PROGRAM C20_ProfinetDrivesCtrl
VAR

	(*G_xLabellerSemaLock	: BOOL;		(* This needs to be used to make sure only 1 client is using the FB instance *)

	fbParameterDisplay		: ARRAY[1..cMAX_PROFINET_DRIVES] OF FB_ParameterDisplayWrapper;
							aProfiNetDrives         : ARRAY[1..cMAX_PROFINET_DRIVES] OF ST_ParameterControl;____					
	xModuleIsActive			: ARRAY[1..cMAX_PROFINET_DRIVES] OF BOOL;*)

	fbProfinetCtrl			: ARRAY[1..cMAX_PROFINET_DRIVES] OF FB_G120Simple_V001;

(*dummy sturcture to be replaced by global PROFINET struct once implemnted*)
{library private}
	stEmptyDriveIn								: ST_DRIVE_INPUT;
	stEmptyDriveOut								: ST_DRIVE_OUTPUT;
	nNoCheckPNetIoError							: UINT;
END_VAR
VAR // added by the converter: edge detectors and wires of the graphical bodies
    _w1, _w2 : BOOL;
END_VAR

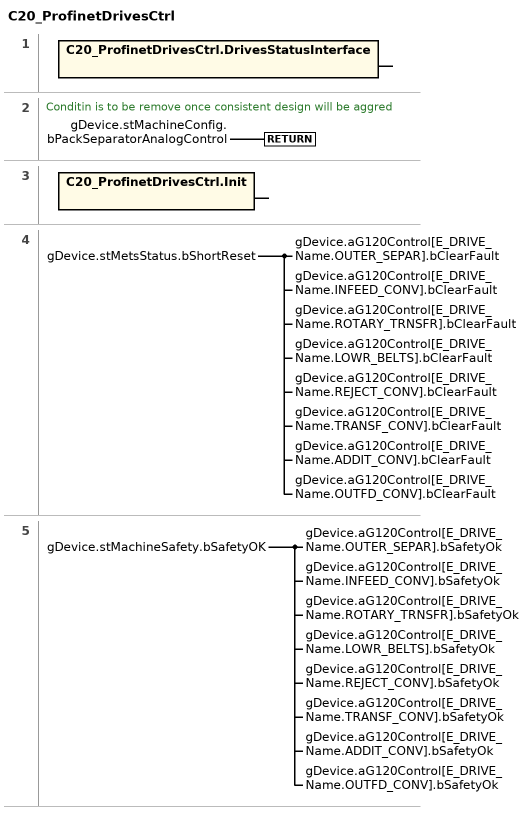
// NETWORK 1
C20_ProfinetDrivesCtrl.DrivesStatusInterface();

// NETWORK 2
// Conditin is to be remove once consistent design will be aggred
IF gDevice.stMachineConfig.bPackSeparatorAnalogControl THEN RETURN; END_IF

// NETWORK 3
C20_ProfinetDrivesCtrl.Init();

// NETWORK 4
_w1 := gDevice.stMetsStatus.bShortReset;
gDevice.aG120Control[E_DRIVE_Name.OUTER_SEPAR].bClearFault := _w1;
gDevice.aG120Control[E_DRIVE_Name.INFEED_CONV].bClearFault := _w1;
gDevice.aG120Control[E_DRIVE_Name.ROTARY_TRNSFR].bClearFault := _w1;
gDevice.aG120Control[E_DRIVE_Name.LOWR_BELTS].bClearFault := _w1;
gDevice.aG120Control[E_DRIVE_Name.REJECT_CONV].bClearFault := _w1;
gDevice.aG120Control[E_DRIVE_Name.TRANSF_CONV].bClearFault := _w1;
gDevice.aG120Control[E_DRIVE_Name.ADDIT_CONV].bClearFault := _w1;
gDevice.aG120Control[E_DRIVE_Name.OUTFD_CONV].bClearFault := _w1;

// NETWORK 5
_w2 := gDevice.stMachineSafety.bSafetyOK;
gDevice.aG120Control[E_DRIVE_Name.OUTER_SEPAR].bSafetyOk := _w2;
gDevice.aG120Control[E_DRIVE_Name.INFEED_CONV].bSafetyOk := _w2;
gDevice.aG120Control[E_DRIVE_Name.ROTARY_TRNSFR].bSafetyOk := _w2;
gDevice.aG120Control[E_DRIVE_Name.LOWR_BELTS].bSafetyOk := _w2;
gDevice.aG120Control[E_DRIVE_Name.REJECT_CONV].bSafetyOk := _w2;
gDevice.aG120Control[E_DRIVE_Name.TRANSF_CONV].bSafetyOk := _w2;
gDevice.aG120Control[E_DRIVE_Name.ADDIT_CONV].bSafetyOk := _w2;
gDevice.aG120Control[E_DRIVE_Name.OUTFD_CONV].bSafetyOk := _w2;

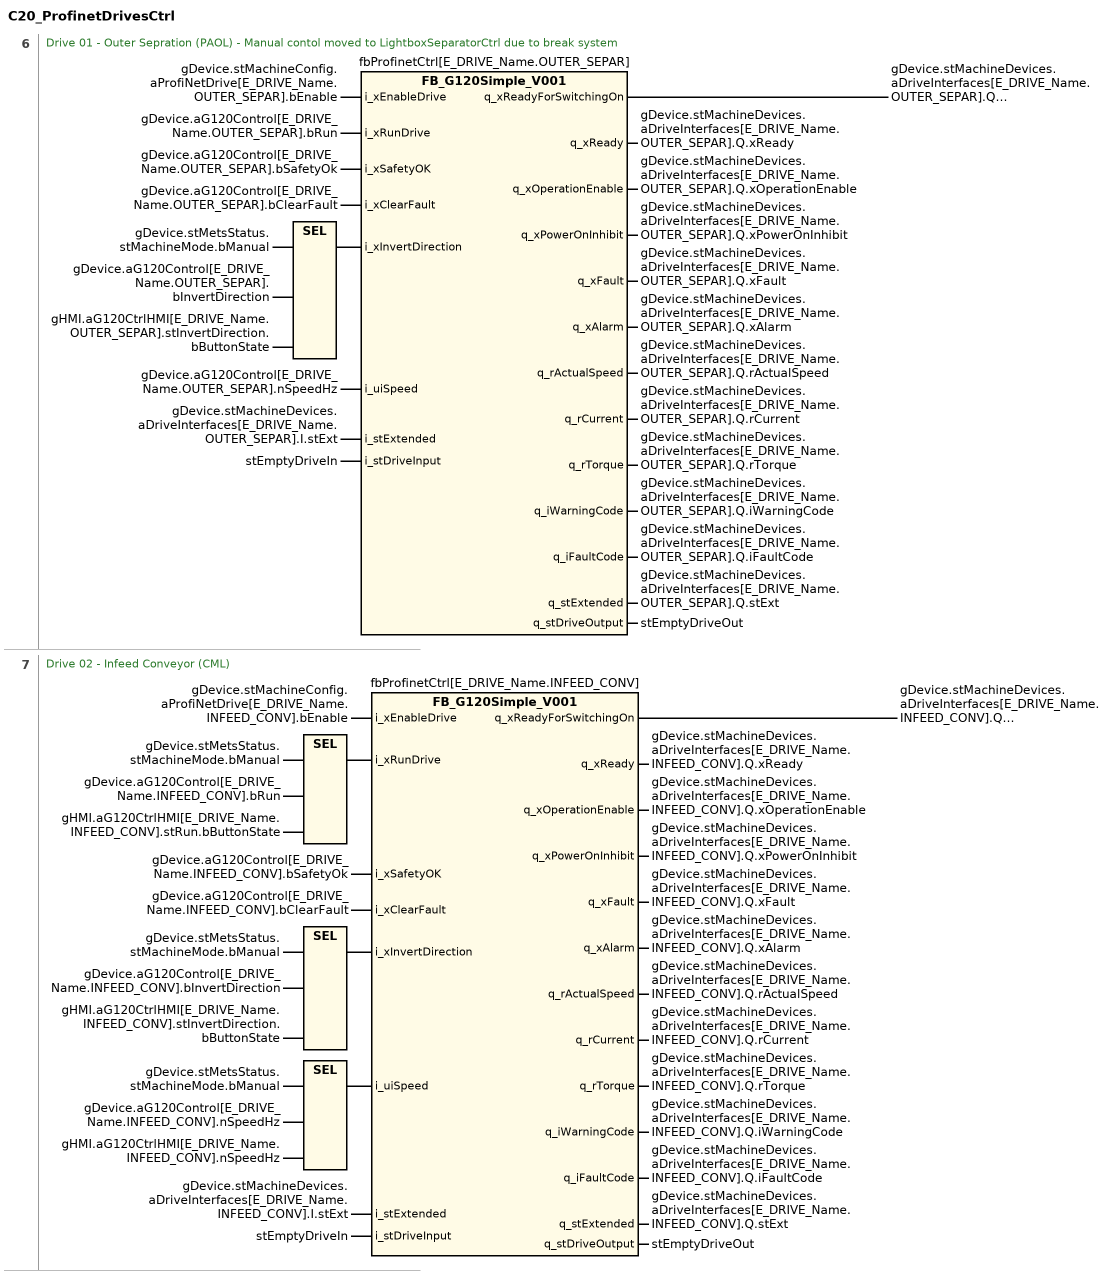
// NETWORK 6
// Drive 01 - Outer Sepration (PAOL) - Manual contol moved to LightboxSeparatorCtrl due to break system
fbProfinetCtrl[E_DRIVE_Name.OUTER_SEPAR](
    i_xEnableDrive := gDevice.stMachineConfig.aProfiNetDrive[E_DRIVE_Name.OUTER_SEPAR].bEnable,
    i_xRunDrive := gDevice.aG120Control[E_DRIVE_Name.OUTER_SEPAR].bRun,
    i_xSafetyOK := gDevice.aG120Control[E_DRIVE_Name.OUTER_SEPAR].bSafetyOk,
    i_xClearFault := gDevice.aG120Control[E_DRIVE_Name.OUTER_SEPAR].bClearFault,
    i_xInvertDirection := SEL(gDevice.stMetsStatus.stMachineMode.bManual, gDevice.aG120Control[E_DRIVE_Name.OUTER_SEPAR].bInvertDirection, gHMI.aG120CtrlHMI[E_DRIVE_Name.OUTER_SEPAR].stInvertDirection.bButtonState),
    i_uiSpeed := gDevice.aG120Control[E_DRIVE_Name.OUTER_SEPAR].nSpeedHz,
    i_stExtended := gDevice.stMachineDevices.aDriveInterfaces[E_DRIVE_Name.OUTER_SEPAR].I.stExt,
    i_stDriveInput := stEmptyDriveIn,
    q_xReady => gDevice.stMachineDevices.aDriveInterfaces[E_DRIVE_Name.OUTER_SEPAR].Q.xReady,
    q_xOperationEnable => gDevice.stMachineDevices.aDriveInterfaces[E_DRIVE_Name.OUTER_SEPAR].Q.xOperationEnable,
    q_xPowerOnInhibit => gDevice.stMachineDevices.aDriveInterfaces[E_DRIVE_Name.OUTER_SEPAR].Q.xPowerOnInhibit,
    q_xFault => gDevice.stMachineDevices.aDriveInterfaces[E_DRIVE_Name.OUTER_SEPAR].Q.xFault,
    q_xAlarm => gDevice.stMachineDevices.aDriveInterfaces[E_DRIVE_Name.OUTER_SEPAR].Q.xAlarm,
    q_rActualSpeed => gDevice.stMachineDevices.aDriveInterfaces[E_DRIVE_Name.OUTER_SEPAR].Q.rActualSpeed,
    q_rCurrent => gDevice.stMachineDevices.aDriveInterfaces[E_DRIVE_Name.OUTER_SEPAR].Q.rCurrent,
    q_rTorque => gDevice.stMachineDevices.aDriveInterfaces[E_DRIVE_Name.OUTER_SEPAR].Q.rTorque,
    q_iWarningCode => gDevice.stMachineDevices.aDriveInterfaces[E_DRIVE_Name.OUTER_SEPAR].Q.iWarningCode,
    q_iFaultCode => gDevice.stMachineDevices.aDriveInterfaces[E_DRIVE_Name.OUTER_SEPAR].Q.iFaultCode,
    q_stExtended => gDevice.stMachineDevices.aDriveInterfaces[E_DRIVE_Name.OUTER_SEPAR].Q.stExt,
    q_stDriveOutput => stEmptyDriveOut); // FB_G120Simple_V001
gDevice.stMachineDevices.aDriveInterfaces[E_DRIVE_Name.OUTER_SEPAR].Q.xReadyForSwitchingOn := fbProfinetCtrl[E_DRIVE_Name.OUTER_SEPAR].q_xReadyForSwitchingOn;

// NETWORK 7
// Drive 02 - Infeed Conveyor (CML)
fbProfinetCtrl[E_DRIVE_Name.INFEED_CONV](
    i_xEnableDrive := gDevice.stMachineConfig.aProfiNetDrive[E_DRIVE_Name.INFEED_CONV].bEnable,
    i_xRunDrive := SEL(gDevice.stMetsStatus.stMachineMode.bManual, gDevice.aG120Control[E_DRIVE_Name.INFEED_CONV].bRun, gHMI.aG120CtrlHMI[E_DRIVE_Name.INFEED_CONV].stRun.bButtonState),
    i_xSafetyOK := gDevice.aG120Control[E_DRIVE_Name.INFEED_CONV].bSafetyOk,
    i_xClearFault := gDevice.aG120Control[E_DRIVE_Name.INFEED_CONV].bClearFault,
    i_xInvertDirection := SEL(gDevice.stMetsStatus.stMachineMode.bManual, gDevice.aG120Control[E_DRIVE_Name.INFEED_CONV].bInvertDirection, gHMI.aG120CtrlHMI[E_DRIVE_Name.INFEED_CONV].stInvertDirection.bButtonState),
    i_uiSpeed := SEL(gDevice.stMetsStatus.stMachineMode.bManual, gDevice.aG120Control[E_DRIVE_Name.INFEED_CONV].nSpeedHz, gHMI.aG120CtrlHMI[E_DRIVE_Name.INFEED_CONV].nSpeedHz),
    i_stExtended := gDevice.stMachineDevices.aDriveInterfaces[E_DRIVE_Name.INFEED_CONV].I.stExt,
    i_stDriveInput := stEmptyDriveIn,
    q_xReady => gDevice.stMachineDevices.aDriveInterfaces[E_DRIVE_Name.INFEED_CONV].Q.xReady,
    q_xOperationEnable => gDevice.stMachineDevices.aDriveInterfaces[E_DRIVE_Name.INFEED_CONV].Q.xOperationEnable,
    q_xPowerOnInhibit => gDevice.stMachineDevices.aDriveInterfaces[E_DRIVE_Name.INFEED_CONV].Q.xPowerOnInhibit,
    q_xFault => gDevice.stMachineDevices.aDriveInterfaces[E_DRIVE_Name.INFEED_CONV].Q.xFault,
    q_xAlarm => gDevice.stMachineDevices.aDriveInterfaces[E_DRIVE_Name.INFEED_CONV].Q.xAlarm,
    q_rActualSpeed => gDevice.stMachineDevices.aDriveInterfaces[E_DRIVE_Name.INFEED_CONV].Q.rActualSpeed,
    q_rCurrent => gDevice.stMachineDevices.aDriveInterfaces[E_DRIVE_Name.INFEED_CONV].Q.rCurrent,
    q_rTorque => gDevice.stMachineDevices.aDriveInterfaces[E_DRIVE_Name.INFEED_CONV].Q.rTorque,
    q_iWarningCode => gDevice.stMachineDevices.aDriveInterfaces[E_DRIVE_Name.INFEED_CONV].Q.iWarningCode,
    q_iFaultCode => gDevice.stMachineDevices.aDriveInterfaces[E_DRIVE_Name.INFEED_CONV].Q.iFaultCode,
    q_stExtended => gDevice.stMachineDevices.aDriveInterfaces[E_DRIVE_Name.INFEED_CONV].Q.stExt,
    q_stDriveOutput => stEmptyDriveOut); // FB_G120Simple_V001
gDevice.stMachineDevices.aDriveInterfaces[E_DRIVE_Name.INFEED_CONV].Q.xReadyForSwitchingOn := fbProfinetCtrl[E_DRIVE_Name.INFEED_CONV].q_xReadyForSwitchingOn;

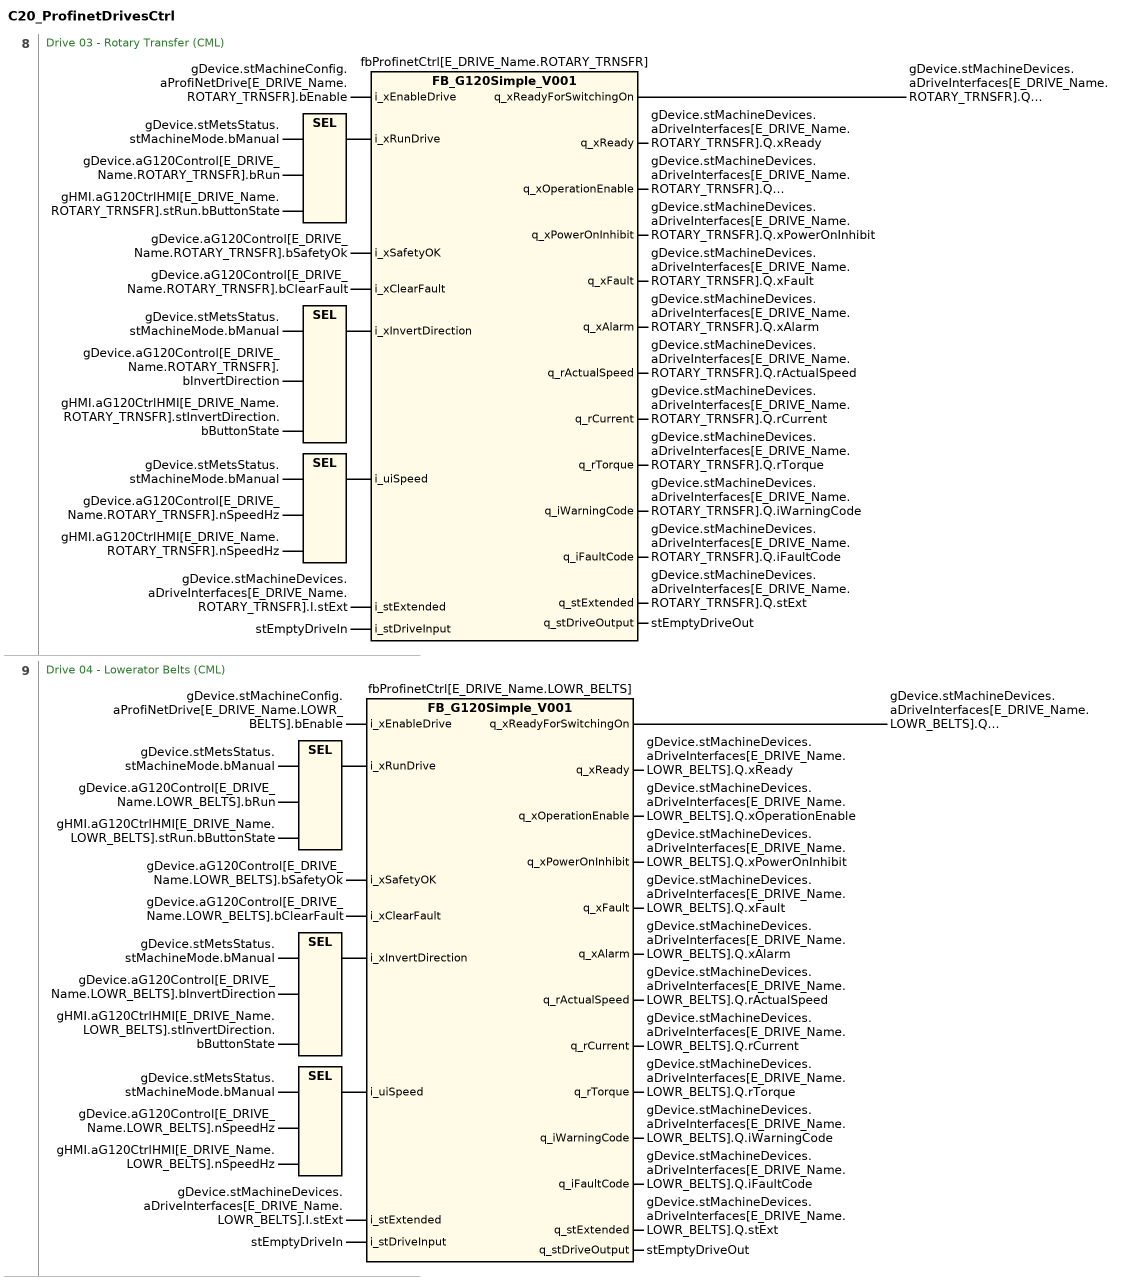
// NETWORK 8
// Drive 03 - Rotary Transfer (CML)
fbProfinetCtrl[E_DRIVE_Name.ROTARY_TRNSFR](
    i_xEnableDrive := gDevice.stMachineConfig.aProfiNetDrive[E_DRIVE_Name.ROTARY_TRNSFR].bEnable,
    i_xRunDrive := SEL(gDevice.stMetsStatus.stMachineMode.bManual, gDevice.aG120Control[E_DRIVE_Name.ROTARY_TRNSFR].bRun, gHMI.aG120CtrlHMI[E_DRIVE_Name.ROTARY_TRNSFR].stRun.bButtonState),
    i_xSafetyOK := gDevice.aG120Control[E_DRIVE_Name.ROTARY_TRNSFR].bSafetyOk,
    i_xClearFault := gDevice.aG120Control[E_DRIVE_Name.ROTARY_TRNSFR].bClearFault,
    i_xInvertDirection := SEL(gDevice.stMetsStatus.stMachineMode.bManual, gDevice.aG120Control[E_DRIVE_Name.ROTARY_TRNSFR].bInvertDirection, gHMI.aG120CtrlHMI[E_DRIVE_Name.ROTARY_TRNSFR].stInvertDirection.bButtonState),
    i_uiSpeed := SEL(gDevice.stMetsStatus.stMachineMode.bManual, gDevice.aG120Control[E_DRIVE_Name.ROTARY_TRNSFR].nSpeedHz, gHMI.aG120CtrlHMI[E_DRIVE_Name.ROTARY_TRNSFR].nSpeedHz),
    i_stExtended := gDevice.stMachineDevices.aDriveInterfaces[E_DRIVE_Name.ROTARY_TRNSFR].I.stExt,
    i_stDriveInput := stEmptyDriveIn,
    q_xReady => gDevice.stMachineDevices.aDriveInterfaces[E_DRIVE_Name.ROTARY_TRNSFR].Q.xReady,
    q_xOperationEnable => gDevice.stMachineDevices.aDriveInterfaces[E_DRIVE_Name.ROTARY_TRNSFR].Q.xOperationEnable,
    q_xPowerOnInhibit => gDevice.stMachineDevices.aDriveInterfaces[E_DRIVE_Name.ROTARY_TRNSFR].Q.xPowerOnInhibit,
    q_xFault => gDevice.stMachineDevices.aDriveInterfaces[E_DRIVE_Name.ROTARY_TRNSFR].Q.xFault,
    q_xAlarm => gDevice.stMachineDevices.aDriveInterfaces[E_DRIVE_Name.ROTARY_TRNSFR].Q.xAlarm,
    q_rActualSpeed => gDevice.stMachineDevices.aDriveInterfaces[E_DRIVE_Name.ROTARY_TRNSFR].Q.rActualSpeed,
    q_rCurrent => gDevice.stMachineDevices.aDriveInterfaces[E_DRIVE_Name.ROTARY_TRNSFR].Q.rCurrent,
    q_rTorque => gDevice.stMachineDevices.aDriveInterfaces[E_DRIVE_Name.ROTARY_TRNSFR].Q.rTorque,
    q_iWarningCode => gDevice.stMachineDevices.aDriveInterfaces[E_DRIVE_Name.ROTARY_TRNSFR].Q.iWarningCode,
    q_iFaultCode => gDevice.stMachineDevices.aDriveInterfaces[E_DRIVE_Name.ROTARY_TRNSFR].Q.iFaultCode,
    q_stExtended => gDevice.stMachineDevices.aDriveInterfaces[E_DRIVE_Name.ROTARY_TRNSFR].Q.stExt,
    q_stDriveOutput => stEmptyDriveOut); // FB_G120Simple_V001
gDevice.stMachineDevices.aDriveInterfaces[E_DRIVE_Name.ROTARY_TRNSFR].Q.xReadyForSwitchingOn := fbProfinetCtrl[E_DRIVE_Name.ROTARY_TRNSFR].q_xReadyForSwitchingOn;

// NETWORK 9
// Drive 04 - Lowerator Belts (CML)
fbProfinetCtrl[E_DRIVE_Name.LOWR_BELTS](
    i_xEnableDrive := gDevice.stMachineConfig.aProfiNetDrive[E_DRIVE_Name.LOWR_BELTS].bEnable,
    i_xRunDrive := SEL(gDevice.stMetsStatus.stMachineMode.bManual, gDevice.aG120Control[E_DRIVE_Name.LOWR_BELTS].bRun, gHMI.aG120CtrlHMI[E_DRIVE_Name.LOWR_BELTS].stRun.bButtonState),
    i_xSafetyOK := gDevice.aG120Control[E_DRIVE_Name.LOWR_BELTS].bSafetyOk,
    i_xClearFault := gDevice.aG120Control[E_DRIVE_Name.LOWR_BELTS].bClearFault,
    i_xInvertDirection := SEL(gDevice.stMetsStatus.stMachineMode.bManual, gDevice.aG120Control[E_DRIVE_Name.LOWR_BELTS].bInvertDirection, gHMI.aG120CtrlHMI[E_DRIVE_Name.LOWR_BELTS].stInvertDirection.bButtonState),
    i_uiSpeed := SEL(gDevice.stMetsStatus.stMachineMode.bManual, gDevice.aG120Control[E_DRIVE_Name.LOWR_BELTS].nSpeedHz, gHMI.aG120CtrlHMI[E_DRIVE_Name.LOWR_BELTS].nSpeedHz),
    i_stExtended := gDevice.stMachineDevices.aDriveInterfaces[E_DRIVE_Name.LOWR_BELTS].I.stExt,
    i_stDriveInput := stEmptyDriveIn,
    q_xReady => gDevice.stMachineDevices.aDriveInterfaces[E_DRIVE_Name.LOWR_BELTS].Q.xReady,
    q_xOperationEnable => gDevice.stMachineDevices.aDriveInterfaces[E_DRIVE_Name.LOWR_BELTS].Q.xOperationEnable,
    q_xPowerOnInhibit => gDevice.stMachineDevices.aDriveInterfaces[E_DRIVE_Name.LOWR_BELTS].Q.xPowerOnInhibit,
    q_xFault => gDevice.stMachineDevices.aDriveInterfaces[E_DRIVE_Name.LOWR_BELTS].Q.xFault,
    q_xAlarm => gDevice.stMachineDevices.aDriveInterfaces[E_DRIVE_Name.LOWR_BELTS].Q.xAlarm,
    q_rActualSpeed => gDevice.stMachineDevices.aDriveInterfaces[E_DRIVE_Name.LOWR_BELTS].Q.rActualSpeed,
    q_rCurrent => gDevice.stMachineDevices.aDriveInterfaces[E_DRIVE_Name.LOWR_BELTS].Q.rCurrent,
    q_rTorque => gDevice.stMachineDevices.aDriveInterfaces[E_DRIVE_Name.LOWR_BELTS].Q.rTorque,
    q_iWarningCode => gDevice.stMachineDevices.aDriveInterfaces[E_DRIVE_Name.LOWR_BELTS].Q.iWarningCode,
    q_iFaultCode => gDevice.stMachineDevices.aDriveInterfaces[E_DRIVE_Name.LOWR_BELTS].Q.iFaultCode,
    q_stExtended => gDevice.stMachineDevices.aDriveInterfaces[E_DRIVE_Name.LOWR_BELTS].Q.stExt,
    q_stDriveOutput => stEmptyDriveOut); // FB_G120Simple_V001
gDevice.stMachineDevices.aDriveInterfaces[E_DRIVE_Name.LOWR_BELTS].Q.xReadyForSwitchingOn := fbProfinetCtrl[E_DRIVE_Name.LOWR_BELTS].q_xReadyForSwitchingOn;

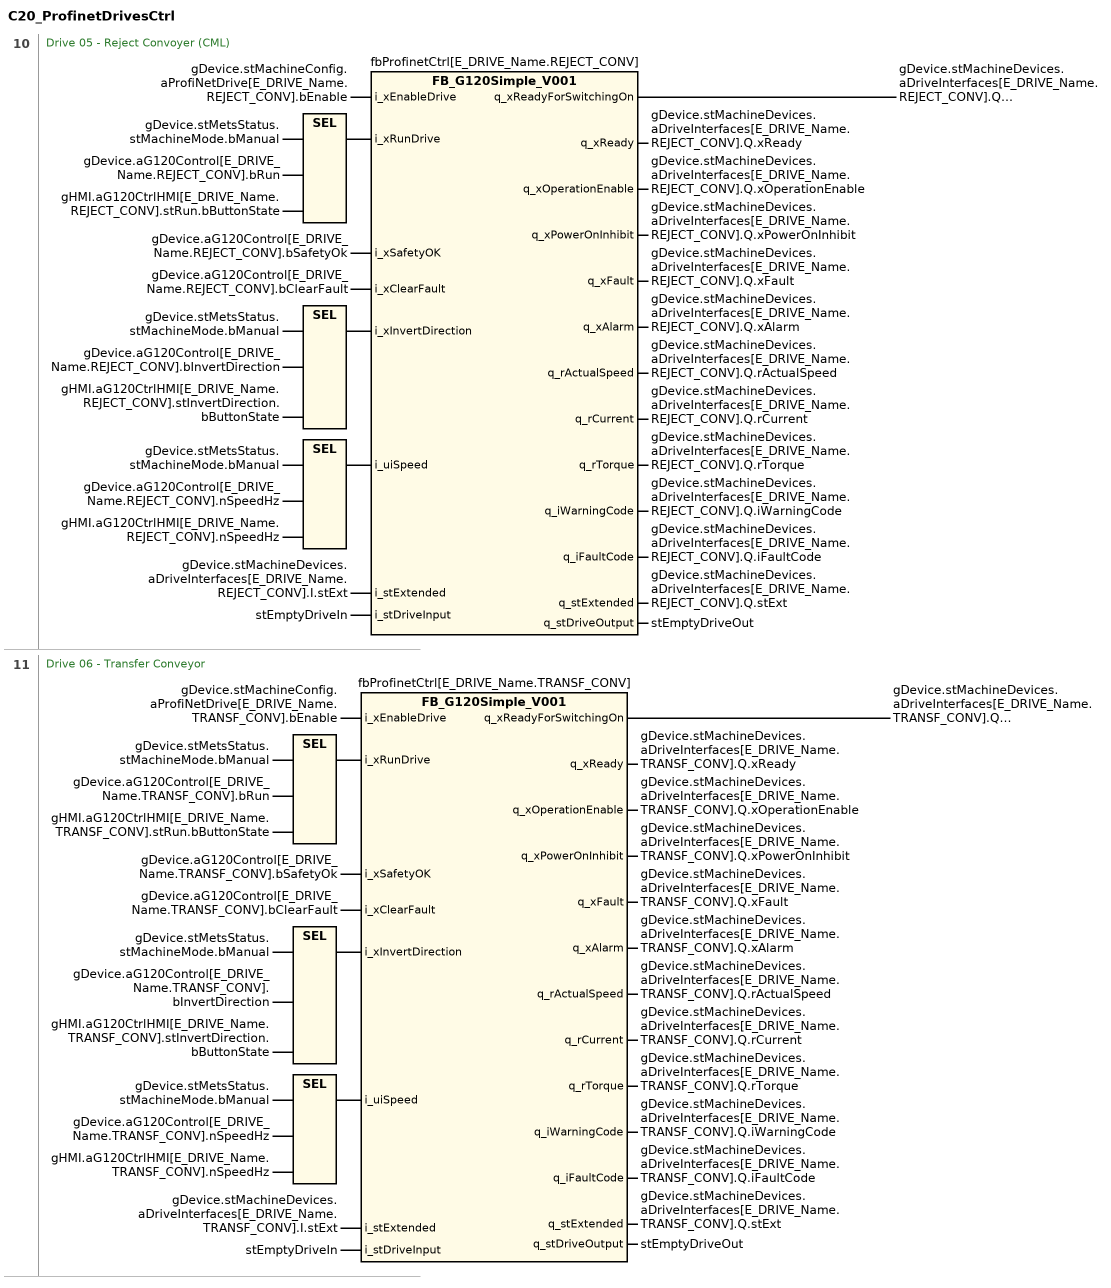
// NETWORK 10
// Drive 05 - Reject Convoyer (CML)
fbProfinetCtrl[E_DRIVE_Name.REJECT_CONV](
    i_xEnableDrive := gDevice.stMachineConfig.aProfiNetDrive[E_DRIVE_Name.REJECT_CONV].bEnable,
    i_xRunDrive := SEL(gDevice.stMetsStatus.stMachineMode.bManual, gDevice.aG120Control[E_DRIVE_Name.REJECT_CONV].bRun, gHMI.aG120CtrlHMI[E_DRIVE_Name.REJECT_CONV].stRun.bButtonState),
    i_xSafetyOK := gDevice.aG120Control[E_DRIVE_Name.REJECT_CONV].bSafetyOk,
    i_xClearFault := gDevice.aG120Control[E_DRIVE_Name.REJECT_CONV].bClearFault,
    i_xInvertDirection := SEL(gDevice.stMetsStatus.stMachineMode.bManual, gDevice.aG120Control[E_DRIVE_Name.REJECT_CONV].bInvertDirection, gHMI.aG120CtrlHMI[E_DRIVE_Name.REJECT_CONV].stInvertDirection.bButtonState),
    i_uiSpeed := SEL(gDevice.stMetsStatus.stMachineMode.bManual, gDevice.aG120Control[E_DRIVE_Name.REJECT_CONV].nSpeedHz, gHMI.aG120CtrlHMI[E_DRIVE_Name.REJECT_CONV].nSpeedHz),
    i_stExtended := gDevice.stMachineDevices.aDriveInterfaces[E_DRIVE_Name.REJECT_CONV].I.stExt,
    i_stDriveInput := stEmptyDriveIn,
    q_xReady => gDevice.stMachineDevices.aDriveInterfaces[E_DRIVE_Name.REJECT_CONV].Q.xReady,
    q_xOperationEnable => gDevice.stMachineDevices.aDriveInterfaces[E_DRIVE_Name.REJECT_CONV].Q.xOperationEnable,
    q_xPowerOnInhibit => gDevice.stMachineDevices.aDriveInterfaces[E_DRIVE_Name.REJECT_CONV].Q.xPowerOnInhibit,
    q_xFault => gDevice.stMachineDevices.aDriveInterfaces[E_DRIVE_Name.REJECT_CONV].Q.xFault,
    q_xAlarm => gDevice.stMachineDevices.aDriveInterfaces[E_DRIVE_Name.REJECT_CONV].Q.xAlarm,
    q_rActualSpeed => gDevice.stMachineDevices.aDriveInterfaces[E_DRIVE_Name.REJECT_CONV].Q.rActualSpeed,
    q_rCurrent => gDevice.stMachineDevices.aDriveInterfaces[E_DRIVE_Name.REJECT_CONV].Q.rCurrent,
    q_rTorque => gDevice.stMachineDevices.aDriveInterfaces[E_DRIVE_Name.REJECT_CONV].Q.rTorque,
    q_iWarningCode => gDevice.stMachineDevices.aDriveInterfaces[E_DRIVE_Name.REJECT_CONV].Q.iWarningCode,
    q_iFaultCode => gDevice.stMachineDevices.aDriveInterfaces[E_DRIVE_Name.REJECT_CONV].Q.iFaultCode,
    q_stExtended => gDevice.stMachineDevices.aDriveInterfaces[E_DRIVE_Name.REJECT_CONV].Q.stExt,
    q_stDriveOutput => stEmptyDriveOut); // FB_G120Simple_V001
gDevice.stMachineDevices.aDriveInterfaces[E_DRIVE_Name.REJECT_CONV].Q.xReadyForSwitchingOn := fbProfinetCtrl[E_DRIVE_Name.REJECT_CONV].q_xReadyForSwitchingOn;

// NETWORK 11
// Drive 06 - Transfer Conveyor
fbProfinetCtrl[E_DRIVE_Name.TRANSF_CONV](
    i_xEnableDrive := gDevice.stMachineConfig.aProfiNetDrive[E_DRIVE_Name.TRANSF_CONV].bEnable,
    i_xRunDrive := SEL(gDevice.stMetsStatus.stMachineMode.bManual, gDevice.aG120Control[E_DRIVE_Name.TRANSF_CONV].bRun, gHMI.aG120CtrlHMI[E_DRIVE_Name.TRANSF_CONV].stRun.bButtonState),
    i_xSafetyOK := gDevice.aG120Control[E_DRIVE_Name.TRANSF_CONV].bSafetyOk,
    i_xClearFault := gDevice.aG120Control[E_DRIVE_Name.TRANSF_CONV].bClearFault,
    i_xInvertDirection := SEL(gDevice.stMetsStatus.stMachineMode.bManual, gDevice.aG120Control[E_DRIVE_Name.TRANSF_CONV].bInvertDirection, gHMI.aG120CtrlHMI[E_DRIVE_Name.TRANSF_CONV].stInvertDirection.bButtonState),
    i_uiSpeed := SEL(gDevice.stMetsStatus.stMachineMode.bManual, gDevice.aG120Control[E_DRIVE_Name.TRANSF_CONV].nSpeedHz, gHMI.aG120CtrlHMI[E_DRIVE_Name.TRANSF_CONV].nSpeedHz),
    i_stExtended := gDevice.stMachineDevices.aDriveInterfaces[E_DRIVE_Name.TRANSF_CONV].I.stExt,
    i_stDriveInput := stEmptyDriveIn,
    q_xReady => gDevice.stMachineDevices.aDriveInterfaces[E_DRIVE_Name.TRANSF_CONV].Q.xReady,
    q_xOperationEnable => gDevice.stMachineDevices.aDriveInterfaces[E_DRIVE_Name.TRANSF_CONV].Q.xOperationEnable,
    q_xPowerOnInhibit => gDevice.stMachineDevices.aDriveInterfaces[E_DRIVE_Name.TRANSF_CONV].Q.xPowerOnInhibit,
    q_xFault => gDevice.stMachineDevices.aDriveInterfaces[E_DRIVE_Name.TRANSF_CONV].Q.xFault,
    q_xAlarm => gDevice.stMachineDevices.aDriveInterfaces[E_DRIVE_Name.TRANSF_CONV].Q.xAlarm,
    q_rActualSpeed => gDevice.stMachineDevices.aDriveInterfaces[E_DRIVE_Name.TRANSF_CONV].Q.rActualSpeed,
    q_rCurrent => gDevice.stMachineDevices.aDriveInterfaces[E_DRIVE_Name.TRANSF_CONV].Q.rCurrent,
    q_rTorque => gDevice.stMachineDevices.aDriveInterfaces[E_DRIVE_Name.TRANSF_CONV].Q.rTorque,
    q_iWarningCode => gDevice.stMachineDevices.aDriveInterfaces[E_DRIVE_Name.TRANSF_CONV].Q.iWarningCode,
    q_iFaultCode => gDevice.stMachineDevices.aDriveInterfaces[E_DRIVE_Name.TRANSF_CONV].Q.iFaultCode,
    q_stExtended => gDevice.stMachineDevices.aDriveInterfaces[E_DRIVE_Name.TRANSF_CONV].Q.stExt,
    q_stDriveOutput => stEmptyDriveOut); // FB_G120Simple_V001
gDevice.stMachineDevices.aDriveInterfaces[E_DRIVE_Name.TRANSF_CONV].Q.xReadyForSwitchingOn := fbProfinetCtrl[E_DRIVE_Name.TRANSF_CONV].q_xReadyForSwitchingOn;

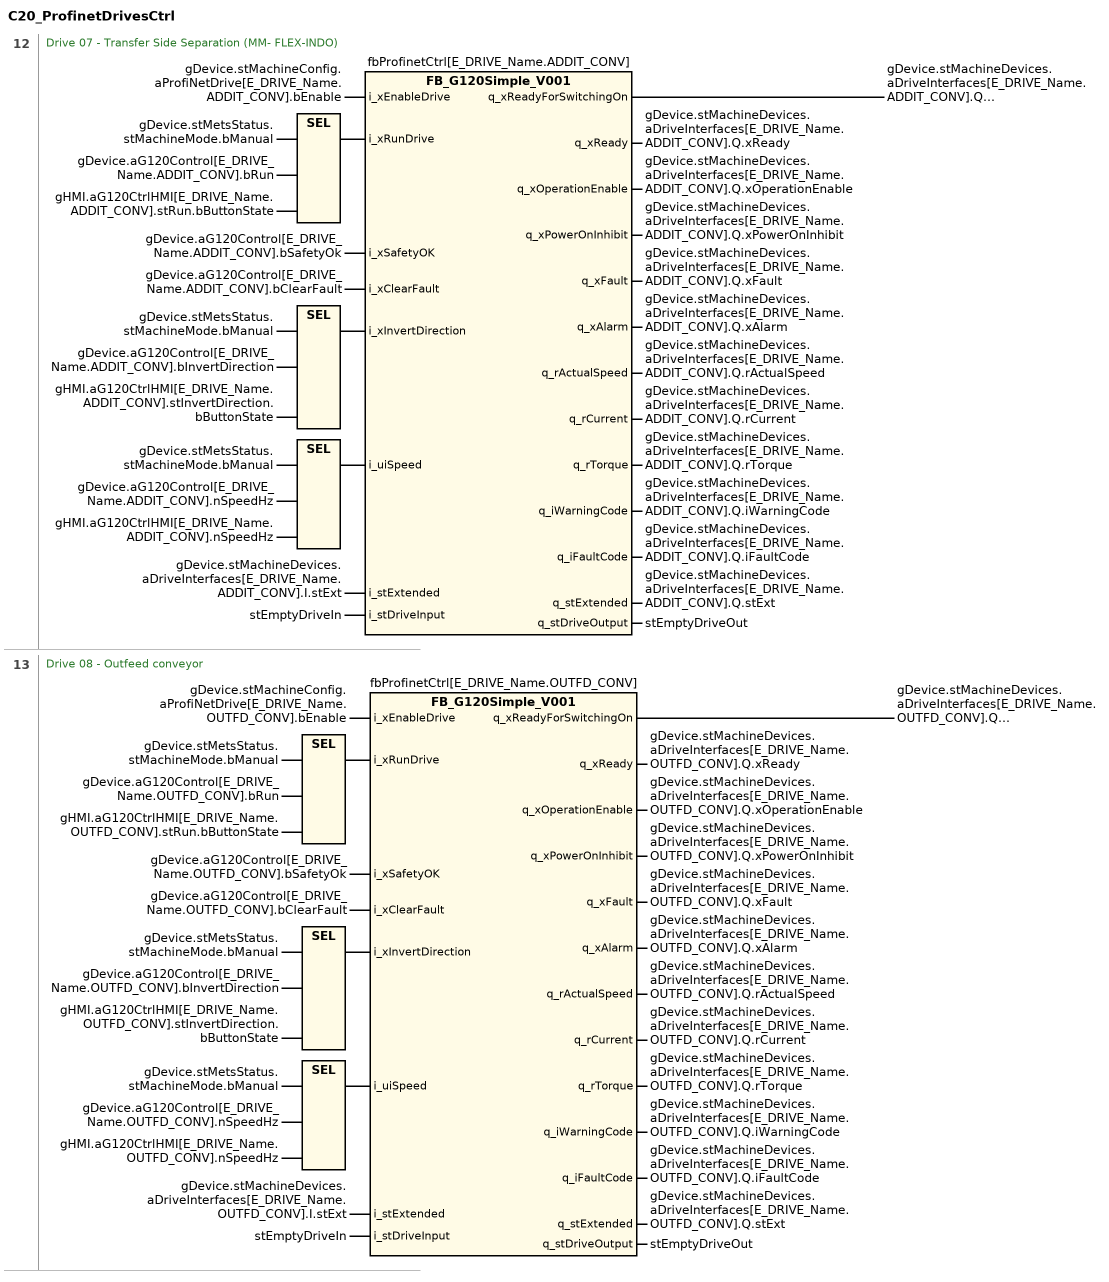
// NETWORK 12
// Drive 07 - Transfer Side Separation (MM- FLEX-INDO)
fbProfinetCtrl[E_DRIVE_Name.ADDIT_CONV](
    i_xEnableDrive := gDevice.stMachineConfig.aProfiNetDrive[E_DRIVE_Name.ADDIT_CONV].bEnable,
    i_xRunDrive := SEL(gDevice.stMetsStatus.stMachineMode.bManual, gDevice.aG120Control[E_DRIVE_Name.ADDIT_CONV].bRun, gHMI.aG120CtrlHMI[E_DRIVE_Name.ADDIT_CONV].stRun.bButtonState),
    i_xSafetyOK := gDevice.aG120Control[E_DRIVE_Name.ADDIT_CONV].bSafetyOk,
    i_xClearFault := gDevice.aG120Control[E_DRIVE_Name.ADDIT_CONV].bClearFault,
    i_xInvertDirection := SEL(gDevice.stMetsStatus.stMachineMode.bManual, gDevice.aG120Control[E_DRIVE_Name.ADDIT_CONV].bInvertDirection, gHMI.aG120CtrlHMI[E_DRIVE_Name.ADDIT_CONV].stInvertDirection.bButtonState),
    i_uiSpeed := SEL(gDevice.stMetsStatus.stMachineMode.bManual, gDevice.aG120Control[E_DRIVE_Name.ADDIT_CONV].nSpeedHz, gHMI.aG120CtrlHMI[E_DRIVE_Name.ADDIT_CONV].nSpeedHz),
    i_stExtended := gDevice.stMachineDevices.aDriveInterfaces[E_DRIVE_Name.ADDIT_CONV].I.stExt,
    i_stDriveInput := stEmptyDriveIn,
    q_xReady => gDevice.stMachineDevices.aDriveInterfaces[E_DRIVE_Name.ADDIT_CONV].Q.xReady,
    q_xOperationEnable => gDevice.stMachineDevices.aDriveInterfaces[E_DRIVE_Name.ADDIT_CONV].Q.xOperationEnable,
    q_xPowerOnInhibit => gDevice.stMachineDevices.aDriveInterfaces[E_DRIVE_Name.ADDIT_CONV].Q.xPowerOnInhibit,
    q_xFault => gDevice.stMachineDevices.aDriveInterfaces[E_DRIVE_Name.ADDIT_CONV].Q.xFault,
    q_xAlarm => gDevice.stMachineDevices.aDriveInterfaces[E_DRIVE_Name.ADDIT_CONV].Q.xAlarm,
    q_rActualSpeed => gDevice.stMachineDevices.aDriveInterfaces[E_DRIVE_Name.ADDIT_CONV].Q.rActualSpeed,
    q_rCurrent => gDevice.stMachineDevices.aDriveInterfaces[E_DRIVE_Name.ADDIT_CONV].Q.rCurrent,
    q_rTorque => gDevice.stMachineDevices.aDriveInterfaces[E_DRIVE_Name.ADDIT_CONV].Q.rTorque,
    q_iWarningCode => gDevice.stMachineDevices.aDriveInterfaces[E_DRIVE_Name.ADDIT_CONV].Q.iWarningCode,
    q_iFaultCode => gDevice.stMachineDevices.aDriveInterfaces[E_DRIVE_Name.ADDIT_CONV].Q.iFaultCode,
    q_stExtended => gDevice.stMachineDevices.aDriveInterfaces[E_DRIVE_Name.ADDIT_CONV].Q.stExt,
    q_stDriveOutput => stEmptyDriveOut); // FB_G120Simple_V001
gDevice.stMachineDevices.aDriveInterfaces[E_DRIVE_Name.ADDIT_CONV].Q.xReadyForSwitchingOn := fbProfinetCtrl[E_DRIVE_Name.ADDIT_CONV].q_xReadyForSwitchingOn;

// NETWORK 13
// Drive 08 - Outfeed conveyor
fbProfinetCtrl[E_DRIVE_Name.OUTFD_CONV](
    i_xEnableDrive := gDevice.stMachineConfig.aProfiNetDrive[E_DRIVE_Name.OUTFD_CONV].bEnable,
    i_xRunDrive := SEL(gDevice.stMetsStatus.stMachineMode.bManual, gDevice.aG120Control[E_DRIVE_Name.OUTFD_CONV].bRun, gHMI.aG120CtrlHMI[E_DRIVE_Name.OUTFD_CONV].stRun.bButtonState),
    i_xSafetyOK := gDevice.aG120Control[E_DRIVE_Name.OUTFD_CONV].bSafetyOk,
    i_xClearFault := gDevice.aG120Control[E_DRIVE_Name.OUTFD_CONV].bClearFault,
    i_xInvertDirection := SEL(gDevice.stMetsStatus.stMachineMode.bManual, gDevice.aG120Control[E_DRIVE_Name.OUTFD_CONV].bInvertDirection, gHMI.aG120CtrlHMI[E_DRIVE_Name.OUTFD_CONV].stInvertDirection.bButtonState),
    i_uiSpeed := SEL(gDevice.stMetsStatus.stMachineMode.bManual, gDevice.aG120Control[E_DRIVE_Name.OUTFD_CONV].nSpeedHz, gHMI.aG120CtrlHMI[E_DRIVE_Name.OUTFD_CONV].nSpeedHz),
    i_stExtended := gDevice.stMachineDevices.aDriveInterfaces[E_DRIVE_Name.OUTFD_CONV].I.stExt,
    i_stDriveInput := stEmptyDriveIn,
    q_xReady => gDevice.stMachineDevices.aDriveInterfaces[E_DRIVE_Name.OUTFD_CONV].Q.xReady,
    q_xOperationEnable => gDevice.stMachineDevices.aDriveInterfaces[E_DRIVE_Name.OUTFD_CONV].Q.xOperationEnable,
    q_xPowerOnInhibit => gDevice.stMachineDevices.aDriveInterfaces[E_DRIVE_Name.OUTFD_CONV].Q.xPowerOnInhibit,
    q_xFault => gDevice.stMachineDevices.aDriveInterfaces[E_DRIVE_Name.OUTFD_CONV].Q.xFault,
    q_xAlarm => gDevice.stMachineDevices.aDriveInterfaces[E_DRIVE_Name.OUTFD_CONV].Q.xAlarm,
    q_rActualSpeed => gDevice.stMachineDevices.aDriveInterfaces[E_DRIVE_Name.OUTFD_CONV].Q.rActualSpeed,
    q_rCurrent => gDevice.stMachineDevices.aDriveInterfaces[E_DRIVE_Name.OUTFD_CONV].Q.rCurrent,
    q_rTorque => gDevice.stMachineDevices.aDriveInterfaces[E_DRIVE_Name.OUTFD_CONV].Q.rTorque,
    q_iWarningCode => gDevice.stMachineDevices.aDriveInterfaces[E_DRIVE_Name.OUTFD_CONV].Q.iWarningCode,
    q_iFaultCode => gDevice.stMachineDevices.aDriveInterfaces[E_DRIVE_Name.OUTFD_CONV].Q.iFaultCode,
    q_stExtended => gDevice.stMachineDevices.aDriveInterfaces[E_DRIVE_Name.OUTFD_CONV].Q.stExt,
    q_stDriveOutput => stEmptyDriveOut); // FB_G120Simple_V001
gDevice.stMachineDevices.aDriveInterfaces[E_DRIVE_Name.OUTFD_CONV].Q.xReadyForSwitchingOn := fbProfinetCtrl[E_DRIVE_Name.OUTFD_CONV].q_xReadyForSwitchingOn;

ACTION DrivesStatusInterface:
(*Drive 01 - Outer Sepration (PAOL)*)

IF NOT gDevice.stMachineSafety.bSafetyOK THEN
	gHMI.aG120CtrlHMI[E_DRIVE_Name.OUTER_SEPAR].stRun.bButtonState := FALSE;
END_IF

gHMI.aG120StatusHMI[E_DRIVE_Name.OUTER_SEPAR].bReadyForSwitchingOn	:=	gDevice.stMachineDevices.aDriveInterfaces[E_DRIVE_Name.OUTER_SEPAR].Q.xReadyForSwitchingOn;
gHMI.aG120StatusHMI[E_DRIVE_Name.OUTER_SEPAR].bReady	:=	gDevice.stMachineDevices.aDriveInterfaces[E_DRIVE_Name.OUTER_SEPAR].Q.xReady;
gHMI.aG120StatusHMI[E_DRIVE_Name.OUTER_SEPAR].bOperationEnable	:=	gDevice.stMachineDevices.aDriveInterfaces[E_DRIVE_Name.OUTER_SEPAR].Q.xOperationEnable;
gHMI.aG120StatusHMI[E_DRIVE_Name.OUTER_SEPAR].bFault	:=	gDevice.stMachineDevices.aDriveInterfaces[E_DRIVE_Name.OUTER_SEPAR].Q.xFault;
gHMI.aG120StatusHMI[E_DRIVE_Name.OUTER_SEPAR].nFaultCode	:=	gDevice.stMachineDevices.aDriveInterfaces[E_DRIVE_Name.OUTER_SEPAR].Q.iFaultCode;
gHMI.aG120StatusHMI[E_DRIVE_Name.OUTER_SEPAR].bAlarm	:=	gDevice.stMachineDevices.aDriveInterfaces[E_DRIVE_Name.OUTER_SEPAR].Q.xAlarm;
gHMI.aG120StatusHMI[E_DRIVE_Name.OUTER_SEPAR].nWarningCode		:=	gDevice.stMachineDevices.aDriveInterfaces[E_DRIVE_Name.OUTER_SEPAR].Q.iWarningCode;
gHMI.aG120StatusHMI[E_DRIVE_Name.OUTER_SEPAR].fActualSpeed	:= gDevice.stMachineDevices.aDriveInterfaces[E_DRIVE_Name.OUTER_SEPAR].Q.rActualSpeed;
gHMI.aG120StatusHMI[E_DRIVE_Name.OUTER_SEPAR].fCurrent	:=	 gDevice.stMachineDevices.aDriveInterfaces[E_DRIVE_Name.OUTER_SEPAR].Q.rCurrent;
gHMI.aG120StatusHMI[E_DRIVE_Name.OUTER_SEPAR].fTorque	:=	 gDevice.stMachineDevices.aDriveInterfaces[E_DRIVE_Name.OUTER_SEPAR].Q.rTorque;
gHMI.aG120StatusHMI[E_DRIVE_Name.OUTER_SEPAR].bTorqueLimitReached		:=  gDevice.stMachineDevices.aDriveInterfaces[E_DRIVE_Name.OUTER_SEPAR].Q.stExt.xTorqueLimitReached;
gHMI.aG120StatusHMI[E_DRIVE_Name.OUTER_SEPAR].bMotorOverTemp	:=  gDevice.stMachineDevices.aDriveInterfaces[E_DRIVE_Name.OUTER_SEPAR].Q.stExt.xMotorOverTemp;
gHMI.aG120StatusHMI[E_DRIVE_Name.OUTER_SEPAR].bHoldingBrake	:=	gDevice.stMachineDevices.aDriveInterfaces[E_DRIVE_Name.OUTER_SEPAR].Q.stExt.xHoldingBrake;

IF (gDevice.stMachineConfig.bPackSeparatorAnalogControl AND NOT gIOFiltered.stPackSeparationDriveOK.bStateInput) OR
	   gDevice.stMachineDevices.aDriveInterfaces[E_DRIVE_Name.OUTER_SEPAR].Q.xFault THEN

	gHMI.aG120StatusHMI[E_DRIVE_Name.OUTER_SEPAR].eDriveStatus			:= E_DRIVE_ERROR;

ELSIF (gDevice.stMachineDevices.aDriverStatus[1].bDriveRun AND gDevice.stMachineDevices.aDriverStatus[1].nDriveAnalog > 0 ) OR
	gDevice.stMachineDevices.aDriveInterfaces[E_DRIVE_Name.OUTER_SEPAR].Q.rActualSpeed > 0	 THEN

	gHMI.aG120StatusHMI[E_DRIVE_Name.OUTER_SEPAR].eDriveStatus			:= E_DRIVE_RUNING;
ELSE
	gHMI.aG120StatusHMI[E_DRIVE_Name.OUTER_SEPAR].eDriveStatus			:= E_DRIVE_SPOPPED;
END_IF

(*Drive 02 - Infeed Conveyor (CML)*)

IF NOT gDevice.stMachineSafety.bSafetyOK THEN
	gHMI.aG120CtrlHMI[E_DRIVE_Name.INFEED_CONV].stRun.bButtonState := FALSE;
END_IF

gHMI.aG120StatusHMI[E_DRIVE_Name.INFEED_CONV].bReadyForSwitchingOn	:=	gDevice.stMachineDevices.aDriveInterfaces[E_DRIVE_Name.INFEED_CONV].Q.xReadyForSwitchingOn;
gHMI.aG120StatusHMI[E_DRIVE_Name.INFEED_CONV].bReady	:=	gDevice.stMachineDevices.aDriveInterfaces[E_DRIVE_Name.INFEED_CONV].Q.xReady;
gHMI.aG120StatusHMI[E_DRIVE_Name.INFEED_CONV].bOperationEnable	:=	gDevice.stMachineDevices.aDriveInterfaces[E_DRIVE_Name.INFEED_CONV].Q.xOperationEnable;
gHMI.aG120StatusHMI[E_DRIVE_Name.INFEED_CONV].bFault	:=	gDevice.stMachineDevices.aDriveInterfaces[E_DRIVE_Name.INFEED_CONV].Q.xFault;
gHMI.aG120StatusHMI[E_DRIVE_Name.INFEED_CONV].nFaultCode	:=	gDevice.stMachineDevices.aDriveInterfaces[E_DRIVE_Name.INFEED_CONV].Q.iFaultCode;
gHMI.aG120StatusHMI[E_DRIVE_Name.INFEED_CONV].bAlarm	:=	gDevice.stMachineDevices.aDriveInterfaces[E_DRIVE_Name.INFEED_CONV].Q.xAlarm;
gHMI.aG120StatusHMI[E_DRIVE_Name.INFEED_CONV].nWarningCode		:=	gDevice.stMachineDevices.aDriveInterfaces[E_DRIVE_Name.INFEED_CONV].Q.iWarningCode;
gHMI.aG120StatusHMI[E_DRIVE_Name.INFEED_CONV].fActualSpeed	:= gDevice.stMachineDevices.aDriveInterfaces[E_DRIVE_Name.INFEED_CONV].Q.rActualSpeed;
gHMI.aG120StatusHMI[E_DRIVE_Name.INFEED_CONV].fCurrent	:=	 gDevice.stMachineDevices.aDriveInterfaces[E_DRIVE_Name.INFEED_CONV].Q.rCurrent;
gHMI.aG120StatusHMI[E_DRIVE_Name.INFEED_CONV].fTorque	:=	 gDevice.stMachineDevices.aDriveInterfaces[E_DRIVE_Name.INFEED_CONV].Q.rTorque;
gHMI.aG120StatusHMI[E_DRIVE_Name.INFEED_CONV].bTorqueLimitReached		:=  gDevice.stMachineDevices.aDriveInterfaces[E_DRIVE_Name.INFEED_CONV].Q.stExt.xTorqueLimitReached;
gHMI.aG120StatusHMI[E_DRIVE_Name.INFEED_CONV].bMotorOverTemp	:=  gDevice.stMachineDevices.aDriveInterfaces[E_DRIVE_Name.INFEED_CONV].Q.stExt.xMotorOverTemp;
gHMI.aG120StatusHMI[E_DRIVE_Name.INFEED_CONV].bHoldingBrake	:=	gDevice.stMachineDevices.aDriveInterfaces[E_DRIVE_Name.INFEED_CONV].Q.stExt.xHoldingBrake;

IF  gDevice.stMachineDevices.aDriveInterfaces[E_DRIVE_Name.INFEED_CONV].Q.xFault THEN

	gHMI.aG120StatusHMI[E_DRIVE_Name.INFEED_CONV].eDriveStatus			:= E_DRIVE_ERROR;

ELSIF gDevice.stMachineDevices.aDriveInterfaces[E_DRIVE_Name.INFEED_CONV].Q.rActualSpeed > 0 THEN

	gHMI.aG120StatusHMI[E_DRIVE_Name.INFEED_CONV].eDriveStatus			:= E_DRIVE_RUNING;
ELSE
	gHMI.aG120StatusHMI[E_DRIVE_Name.INFEED_CONV].eDriveStatus			:= E_DRIVE_SPOPPED;
END_IF

(*Drive 03 - Rotary Transfer (CML)*)

IF NOT gDevice.stMachineSafety.bSafetyOK THEN
	gHMI.aG120CtrlHMI[E_DRIVE_Name.ROTARY_TRNSFR].stRun.bButtonState := FALSE;
END_IF

gHMI.aG120StatusHMI[E_DRIVE_Name.ROTARY_TRNSFR].bReadyForSwitchingOn	:=	gDevice.stMachineDevices.aDriveInterfaces[E_DRIVE_Name.ROTARY_TRNSFR].Q.xReadyForSwitchingOn;
gHMI.aG120StatusHMI[E_DRIVE_Name.ROTARY_TRNSFR].bReady	:=	gDevice.stMachineDevices.aDriveInterfaces[E_DRIVE_Name.ROTARY_TRNSFR].Q.xReady;
gHMI.aG120StatusHMI[E_DRIVE_Name.ROTARY_TRNSFR].bOperationEnable	:=	gDevice.stMachineDevices.aDriveInterfaces[E_DRIVE_Name.ROTARY_TRNSFR].Q.xOperationEnable;
gHMI.aG120StatusHMI[E_DRIVE_Name.ROTARY_TRNSFR].bFault	:=	gDevice.stMachineDevices.aDriveInterfaces[E_DRIVE_Name.ROTARY_TRNSFR].Q.xFault;
gHMI.aG120StatusHMI[E_DRIVE_Name.ROTARY_TRNSFR].nFaultCode	:=	gDevice.stMachineDevices.aDriveInterfaces[E_DRIVE_Name.ROTARY_TRNSFR].Q.iFaultCode;
gHMI.aG120StatusHMI[E_DRIVE_Name.ROTARY_TRNSFR].bAlarm	:=	gDevice.stMachineDevices.aDriveInterfaces[E_DRIVE_Name.ROTARY_TRNSFR].Q.xAlarm;
gHMI.aG120StatusHMI[E_DRIVE_Name.ROTARY_TRNSFR].nWarningCode		:=	gDevice.stMachineDevices.aDriveInterfaces[E_DRIVE_Name.ROTARY_TRNSFR].Q.iWarningCode;
gHMI.aG120StatusHMI[E_DRIVE_Name.ROTARY_TRNSFR].fActualSpeed	:= gDevice.stMachineDevices.aDriveInterfaces[E_DRIVE_Name.ROTARY_TRNSFR].Q.rActualSpeed;
gHMI.aG120StatusHMI[E_DRIVE_Name.ROTARY_TRNSFR].fCurrent	:=	 gDevice.stMachineDevices.aDriveInterfaces[E_DRIVE_Name.ROTARY_TRNSFR].Q.rCurrent;
gHMI.aG120StatusHMI[E_DRIVE_Name.ROTARY_TRNSFR].fTorque	:=	 gDevice.stMachineDevices.aDriveInterfaces[E_DRIVE_Name.ROTARY_TRNSFR].Q.rTorque;
gHMI.aG120StatusHMI[E_DRIVE_Name.ROTARY_TRNSFR].bTorqueLimitReached		:=  gDevice.stMachineDevices.aDriveInterfaces[E_DRIVE_Name.ROTARY_TRNSFR].Q.stExt.xTorqueLimitReached;
gHMI.aG120StatusHMI[E_DRIVE_Name.ROTARY_TRNSFR].bMotorOverTemp	:=  gDevice.stMachineDevices.aDriveInterfaces[E_DRIVE_Name.ROTARY_TRNSFR].Q.stExt.xMotorOverTemp;
gHMI.aG120StatusHMI[E_DRIVE_Name.ROTARY_TRNSFR].bHoldingBrake	:=	gDevice.stMachineDevices.aDriveInterfaces[E_DRIVE_Name.ROTARY_TRNSFR].Q.stExt.xHoldingBrake;

IF  gDevice.stMachineDevices.aDriveInterfaces[E_DRIVE_Name.ROTARY_TRNSFR].Q.xFault THEN

	gHMI.aG120StatusHMI[E_DRIVE_Name.ROTARY_TRNSFR].eDriveStatus			:= E_DRIVE_ERROR;

ELSIF gDevice.stMachineDevices.aDriveInterfaces[E_DRIVE_Name.ROTARY_TRNSFR].Q.rActualSpeed > 0 THEN

	gHMI.aG120StatusHMI[E_DRIVE_Name.ROTARY_TRNSFR].eDriveStatus			:= E_DRIVE_RUNING;
ELSE
	gHMI.aG120StatusHMI[E_DRIVE_Name.ROTARY_TRNSFR].eDriveStatus			:= E_DRIVE_SPOPPED;
END_IF

(*Drive 04 - Lowerator Belts (CML)*)

IF NOT gDevice.stMachineSafety.bSafetyOK THEN
	gHMI.aG120CtrlHMI[E_DRIVE_Name.LOWR_BELTS].stRun.bButtonState := FALSE;
END_IF

gHMI.aG120StatusHMI[E_DRIVE_Name.LOWR_BELTS].bReadyForSwitchingOn	:=	gDevice.stMachineDevices.aDriveInterfaces[E_DRIVE_Name.LOWR_BELTS].Q.xReadyForSwitchingOn;
gHMI.aG120StatusHMI[E_DRIVE_Name.LOWR_BELTS].bReady	:=	gDevice.stMachineDevices.aDriveInterfaces[E_DRIVE_Name.LOWR_BELTS].Q.xReady;
gHMI.aG120StatusHMI[E_DRIVE_Name.LOWR_BELTS].bOperationEnable	:=	gDevice.stMachineDevices.aDriveInterfaces[E_DRIVE_Name.LOWR_BELTS].Q.xOperationEnable;
gHMI.aG120StatusHMI[E_DRIVE_Name.LOWR_BELTS].bFault	:=	gDevice.stMachineDevices.aDriveInterfaces[E_DRIVE_Name.LOWR_BELTS].Q.xFault;
gHMI.aG120StatusHMI[E_DRIVE_Name.LOWR_BELTS].nFaultCode	:=	gDevice.stMachineDevices.aDriveInterfaces[E_DRIVE_Name.LOWR_BELTS].Q.iFaultCode;
gHMI.aG120StatusHMI[E_DRIVE_Name.LOWR_BELTS].bAlarm	:=	gDevice.stMachineDevices.aDriveInterfaces[E_DRIVE_Name.LOWR_BELTS].Q.xAlarm;
gHMI.aG120StatusHMI[E_DRIVE_Name.LOWR_BELTS].nWarningCode		:=	gDevice.stMachineDevices.aDriveInterfaces[E_DRIVE_Name.LOWR_BELTS].Q.iWarningCode;
gHMI.aG120StatusHMI[E_DRIVE_Name.LOWR_BELTS].fActualSpeed	:= gDevice.stMachineDevices.aDriveInterfaces[E_DRIVE_Name.LOWR_BELTS].Q.rActualSpeed;
gHMI.aG120StatusHMI[E_DRIVE_Name.LOWR_BELTS].fCurrent	:=	 gDevice.stMachineDevices.aDriveInterfaces[E_DRIVE_Name.LOWR_BELTS].Q.rCurrent;
gHMI.aG120StatusHMI[E_DRIVE_Name.LOWR_BELTS].fTorque	:=	 gDevice.stMachineDevices.aDriveInterfaces[E_DRIVE_Name.LOWR_BELTS].Q.rTorque;
gHMI.aG120StatusHMI[E_DRIVE_Name.LOWR_BELTS].bTorqueLimitReached		:=  gDevice.stMachineDevices.aDriveInterfaces[E_DRIVE_Name.LOWR_BELTS].Q.stExt.xTorqueLimitReached;
gHMI.aG120StatusHMI[E_DRIVE_Name.LOWR_BELTS].bMotorOverTemp	:=  gDevice.stMachineDevices.aDriveInterfaces[E_DRIVE_Name.LOWR_BELTS].Q.stExt.xMotorOverTemp;
gHMI.aG120StatusHMI[E_DRIVE_Name.LOWR_BELTS].bHoldingBrake	:=	gDevice.stMachineDevices.aDriveInterfaces[E_DRIVE_Name.LOWR_BELTS].Q.stExt.xHoldingBrake;

IF  gDevice.stMachineDevices.aDriveInterfaces[E_DRIVE_Name.LOWR_BELTS].Q.xFault THEN

	gHMI.aG120StatusHMI[E_DRIVE_Name.LOWR_BELTS].eDriveStatus			:= E_DRIVE_ERROR;

ELSIF gDevice.stMachineDevices.aDriveInterfaces[E_DRIVE_Name.LOWR_BELTS].Q.rActualSpeed > 0 THEN

	gHMI.aG120StatusHMI[E_DRIVE_Name.LOWR_BELTS].eDriveStatus			:= E_DRIVE_RUNING;
ELSE
	gHMI.aG120StatusHMI[E_DRIVE_Name.LOWR_BELTS].eDriveStatus			:= E_DRIVE_SPOPPED;
END_IF

(*Drive 05 - Reject Convoyer (CML)*)

IF NOT gDevice.stMachineSafety.bSafetyOK THEN
	gHMI.aG120CtrlHMI[E_DRIVE_Name.REJECT_CONV].stRun.bButtonState := FALSE;
END_IF

gHMI.aG120StatusHMI[E_DRIVE_Name.REJECT_CONV].bReadyForSwitchingOn	:=	gDevice.stMachineDevices.aDriveInterfaces[E_DRIVE_Name.REJECT_CONV].Q.xReadyForSwitchingOn;
gHMI.aG120StatusHMI[E_DRIVE_Name.REJECT_CONV].bReady	:=	gDevice.stMachineDevices.aDriveInterfaces[E_DRIVE_Name.REJECT_CONV].Q.xReady;
gHMI.aG120StatusHMI[E_DRIVE_Name.REJECT_CONV].bOperationEnable	:=	gDevice.stMachineDevices.aDriveInterfaces[E_DRIVE_Name.REJECT_CONV].Q.xOperationEnable;
gHMI.aG120StatusHMI[E_DRIVE_Name.REJECT_CONV].bFault	:=	gDevice.stMachineDevices.aDriveInterfaces[E_DRIVE_Name.REJECT_CONV].Q.xFault;
gHMI.aG120StatusHMI[E_DRIVE_Name.REJECT_CONV].nFaultCode	:=	gDevice.stMachineDevices.aDriveInterfaces[E_DRIVE_Name.REJECT_CONV].Q.iFaultCode;
gHMI.aG120StatusHMI[E_DRIVE_Name.REJECT_CONV].bAlarm	:=	gDevice.stMachineDevices.aDriveInterfaces[E_DRIVE_Name.REJECT_CONV].Q.xAlarm;
gHMI.aG120StatusHMI[E_DRIVE_Name.REJECT_CONV].nWarningCode		:=	gDevice.stMachineDevices.aDriveInterfaces[E_DRIVE_Name.REJECT_CONV].Q.iWarningCode;
gHMI.aG120StatusHMI[E_DRIVE_Name.REJECT_CONV].fActualSpeed	:= gDevice.stMachineDevices.aDriveInterfaces[E_DRIVE_Name.REJECT_CONV].Q.rActualSpeed;
gHMI.aG120StatusHMI[E_DRIVE_Name.REJECT_CONV].fCurrent	:=	 gDevice.stMachineDevices.aDriveInterfaces[E_DRIVE_Name.REJECT_CONV].Q.rCurrent;
gHMI.aG120StatusHMI[E_DRIVE_Name.REJECT_CONV].fTorque	:=	 gDevice.stMachineDevices.aDriveInterfaces[E_DRIVE_Name.REJECT_CONV].Q.rTorque;
gHMI.aG120StatusHMI[E_DRIVE_Name.REJECT_CONV].bTorqueLimitReached		:=  gDevice.stMachineDevices.aDriveInterfaces[E_DRIVE_Name.REJECT_CONV].Q.stExt.xTorqueLimitReached;
gHMI.aG120StatusHMI[E_DRIVE_Name.REJECT_CONV].bMotorOverTemp	:=  gDevice.stMachineDevices.aDriveInterfaces[E_DRIVE_Name.REJECT_CONV].Q.stExt.xMotorOverTemp;
gHMI.aG120StatusHMI[E_DRIVE_Name.REJECT_CONV].bHoldingBrake	:=	gDevice.stMachineDevices.aDriveInterfaces[E_DRIVE_Name.REJECT_CONV].Q.stExt.xHoldingBrake;

IF  gDevice.stMachineDevices.aDriveInterfaces[E_DRIVE_Name.REJECT_CONV].Q.xFault THEN

	gHMI.aG120StatusHMI[E_DRIVE_Name.REJECT_CONV].eDriveStatus			:= E_DRIVE_ERROR;

ELSIF gDevice.stMachineDevices.aDriveInterfaces[E_DRIVE_Name.REJECT_CONV].Q.rActualSpeed > 0 THEN

	gHMI.aG120StatusHMI[E_DRIVE_Name.REJECT_CONV].eDriveStatus			:= E_DRIVE_RUNING;
ELSE
	gHMI.aG120StatusHMI[E_DRIVE_Name.REJECT_CONV].eDriveStatus			:= E_DRIVE_SPOPPED;
END_IF

(*Drive 06 - Transfer Conveyor (MM)*)

IF NOT gDevice.stMachineSafety.bSafetyOK THEN
	gHMI.aG120CtrlHMI[E_DRIVE_Name.TRANSF_CONV].stRun.bButtonState := FALSE;
END_IF

gHMI.aG120StatusHMI[E_DRIVE_Name.TRANSF_CONV].bReadyForSwitchingOn	:=	gDevice.stMachineDevices.aDriveInterfaces[E_DRIVE_Name.TRANSF_CONV].Q.xReadyForSwitchingOn;
gHMI.aG120StatusHMI[E_DRIVE_Name.TRANSF_CONV].bReady	:=	gDevice.stMachineDevices.aDriveInterfaces[E_DRIVE_Name.TRANSF_CONV].Q.xReady;
gHMI.aG120StatusHMI[E_DRIVE_Name.TRANSF_CONV].bOperationEnable	:=	gDevice.stMachineDevices.aDriveInterfaces[E_DRIVE_Name.TRANSF_CONV].Q.xOperationEnable;
gHMI.aG120StatusHMI[E_DRIVE_Name.TRANSF_CONV].bFault	:=	gDevice.stMachineDevices.aDriveInterfaces[E_DRIVE_Name.TRANSF_CONV].Q.xFault;
gHMI.aG120StatusHMI[E_DRIVE_Name.TRANSF_CONV].nFaultCode	:=	gDevice.stMachineDevices.aDriveInterfaces[E_DRIVE_Name.TRANSF_CONV].Q.iFaultCode;
gHMI.aG120StatusHMI[E_DRIVE_Name.TRANSF_CONV].bAlarm	:=	gDevice.stMachineDevices.aDriveInterfaces[E_DRIVE_Name.TRANSF_CONV].Q.xAlarm;
gHMI.aG120StatusHMI[E_DRIVE_Name.TRANSF_CONV].nWarningCode		:=	gDevice.stMachineDevices.aDriveInterfaces[E_DRIVE_Name.TRANSF_CONV].Q.iWarningCode;
gHMI.aG120StatusHMI[E_DRIVE_Name.TRANSF_CONV].fActualSpeed	:= gDevice.stMachineDevices.aDriveInterfaces[E_DRIVE_Name.TRANSF_CONV].Q.rActualSpeed;
gHMI.aG120StatusHMI[E_DRIVE_Name.TRANSF_CONV].fCurrent	:=	 gDevice.stMachineDevices.aDriveInterfaces[E_DRIVE_Name.TRANSF_CONV].Q.rCurrent;
gHMI.aG120StatusHMI[E_DRIVE_Name.TRANSF_CONV].fTorque	:=	 gDevice.stMachineDevices.aDriveInterfaces[E_DRIVE_Name.TRANSF_CONV].Q.rTorque;
gHMI.aG120StatusHMI[E_DRIVE_Name.TRANSF_CONV].bTorqueLimitReached		:=  gDevice.stMachineDevices.aDriveInterfaces[E_DRIVE_Name.TRANSF_CONV].Q.stExt.xTorqueLimitReached;
gHMI.aG120StatusHMI[E_DRIVE_Name.TRANSF_CONV].bMotorOverTemp	:=  gDevice.stMachineDevices.aDriveInterfaces[E_DRIVE_Name.TRANSF_CONV].Q.stExt.xMotorOverTemp;
gHMI.aG120StatusHMI[E_DRIVE_Name.TRANSF_CONV].bHoldingBrake	:=	gDevice.stMachineDevices.aDriveInterfaces[E_DRIVE_Name.TRANSF_CONV].Q.stExt.xHoldingBrake;

IF  gDevice.stMachineDevices.aDriveInterfaces[E_DRIVE_Name.TRANSF_CONV].Q.xFault THEN

	gHMI.aG120StatusHMI[E_DRIVE_Name.TRANSF_CONV].eDriveStatus			:= E_DRIVE_ERROR;

ELSIF gDevice.stMachineDevices.aDriveInterfaces[E_DRIVE_Name.TRANSF_CONV].Q.rActualSpeed > 0 THEN

	gHMI.aG120StatusHMI[E_DRIVE_Name.TRANSF_CONV].eDriveStatus			:= E_DRIVE_RUNING;
ELSE
	gHMI.aG120StatusHMI[E_DRIVE_Name.TRANSF_CONV].eDriveStatus			:= E_DRIVE_SPOPPED;
END_IF

(*Drive 07 - Transfer Side Separation (MM)*)

IF NOT gDevice.stMachineSafety.bSafetyOK THEN
	gHMI.aG120CtrlHMI[E_DRIVE_Name.ADDIT_CONV].stRun.bButtonState := FALSE;
END_IF
gHMI.aG120StatusHMI[E_DRIVE_Name.ADDIT_CONV].bReadyForSwitchingOn	:=	gDevice.stMachineDevices.aDriveInterfaces[E_DRIVE_Name.OUTFD_CONV].Q.xReadyForSwitchingOn;
gHMI.aG120StatusHMI[E_DRIVE_Name.ADDIT_CONV].bReady	:=	gDevice.stMachineDevices.aDriveInterfaces[E_DRIVE_Name.ADDIT_CONV].Q.xReady;
gHMI.aG120StatusHMI[E_DRIVE_Name.ADDIT_CONV].bOperationEnable	:=	gDevice.stMachineDevices.aDriveInterfaces[E_DRIVE_Name.ADDIT_CONV].Q.xOperationEnable;
gHMI.aG120StatusHMI[E_DRIVE_Name.ADDIT_CONV].bFault	:=	gDevice.stMachineDevices.aDriveInterfaces[E_DRIVE_Name.ADDIT_CONV].Q.xFault;
gHMI.aG120StatusHMI[E_DRIVE_Name.ADDIT_CONV].nFaultCode	:=	gDevice.stMachineDevices.aDriveInterfaces[E_DRIVE_Name.ADDIT_CONV].Q.iFaultCode;
gHMI.aG120StatusHMI[E_DRIVE_Name.ADDIT_CONV].bAlarm	:=	gDevice.stMachineDevices.aDriveInterfaces[E_DRIVE_Name.ADDIT_CONV].Q.xAlarm;
gHMI.aG120StatusHMI[E_DRIVE_Name.ADDIT_CONV].nWarningCode		:=	gDevice.stMachineDevices.aDriveInterfaces[E_DRIVE_Name.ADDIT_CONV].Q.iWarningCode;
gHMI.aG120StatusHMI[E_DRIVE_Name.ADDIT_CONV].fActualSpeed	:= gDevice.stMachineDevices.aDriveInterfaces[E_DRIVE_Name.ADDIT_CONV].Q.rActualSpeed;
gHMI.aG120StatusHMI[E_DRIVE_Name.ADDIT_CONV].fCurrent	:=	 gDevice.stMachineDevices.aDriveInterfaces[E_DRIVE_Name.ADDIT_CONV].Q.rCurrent;
gHMI.aG120StatusHMI[E_DRIVE_Name.ADDIT_CONV].fTorque	:=	 gDevice.stMachineDevices.aDriveInterfaces[E_DRIVE_Name.ADDIT_CONV].Q.rTorque;
gHMI.aG120StatusHMI[E_DRIVE_Name.ADDIT_CONV].bTorqueLimitReached		:=  gDevice.stMachineDevices.aDriveInterfaces[E_DRIVE_Name.ADDIT_CONV].Q.stExt.xTorqueLimitReached;
gHMI.aG120StatusHMI[E_DRIVE_Name.ADDIT_CONV].bMotorOverTemp	:=  gDevice.stMachineDevices.aDriveInterfaces[E_DRIVE_Name.ADDIT_CONV].Q.stExt.xMotorOverTemp;
gHMI.aG120StatusHMI[E_DRIVE_Name.ADDIT_CONV].bHoldingBrake	:=	gDevice.stMachineDevices.aDriveInterfaces[E_DRIVE_Name.ADDIT_CONV].Q.stExt.xHoldingBrake;

IF  gDevice.stMachineDevices.aDriveInterfaces[E_DRIVE_Name.ADDIT_CONV].Q.xFault THEN

	gHMI.aG120StatusHMI[E_DRIVE_Name.ADDIT_CONV].eDriveStatus			:= E_DRIVE_ERROR;

ELSIF gDevice.stMachineDevices.aDriveInterfaces[E_DRIVE_Name.ADDIT_CONV].Q.rActualSpeed > 0 THEN

	gHMI.aG120StatusHMI[E_DRIVE_Name.ADDIT_CONV].eDriveStatus			:= E_DRIVE_RUNING;
ELSE
	gHMI.aG120StatusHMI[E_DRIVE_Name.ADDIT_CONV].eDriveStatus			:= E_DRIVE_SPOPPED;
END_IF

(*Drive 08 - Spare*)

IF NOT gDevice.stMachineSafety.bSafetyOK THEN
	gHMI.aG120CtrlHMI[E_DRIVE_Name.OUTFD_CONV].stRun.bButtonState := FALSE;
END_IF

gHMI.aG120StatusHMI[E_DRIVE_Name.OUTFD_CONV].bReadyForSwitchingOn	:=	gDevice.stMachineDevices.aDriveInterfaces[E_DRIVE_Name.OUTFD_CONV].Q.xReadyForSwitchingOn;
gHMI.aG120StatusHMI[E_DRIVE_Name.OUTFD_CONV].bReady	:=	gDevice.stMachineDevices.aDriveInterfaces[E_DRIVE_Name.OUTFD_CONV].Q.xReady;
gHMI.aG120StatusHMI[E_DRIVE_Name.OUTFD_CONV].bOperationEnable	:=	gDevice.stMachineDevices.aDriveInterfaces[E_DRIVE_Name.OUTFD_CONV].Q.xOperationEnable;
gHMI.aG120StatusHMI[E_DRIVE_Name.OUTFD_CONV].bFault	:=	gDevice.stMachineDevices.aDriveInterfaces[E_DRIVE_Name.OUTFD_CONV].Q.xFault;
gHMI.aG120StatusHMI[E_DRIVE_Name.OUTFD_CONV].nFaultCode	:=	gDevice.stMachineDevices.aDriveInterfaces[E_DRIVE_Name.OUTFD_CONV].Q.iFaultCode;
gHMI.aG120StatusHMI[E_DRIVE_Name.OUTFD_CONV].bAlarm	:=	gDevice.stMachineDevices.aDriveInterfaces[E_DRIVE_Name.OUTFD_CONV].Q.xAlarm;
gHMI.aG120StatusHMI[E_DRIVE_Name.OUTFD_CONV].nWarningCode		:=	gDevice.stMachineDevices.aDriveInterfaces[E_DRIVE_Name.OUTFD_CONV].Q.iWarningCode;
gHMI.aG120StatusHMI[E_DRIVE_Name.OUTFD_CONV].fActualSpeed	:= gDevice.stMachineDevices.aDriveInterfaces[E_DRIVE_Name.OUTFD_CONV].Q.rActualSpeed;
gHMI.aG120StatusHMI[E_DRIVE_Name.OUTFD_CONV].fCurrent	:=	 gDevice.stMachineDevices.aDriveInterfaces[E_DRIVE_Name.OUTFD_CONV].Q.rCurrent;
gHMI.aG120StatusHMI[E_DRIVE_Name.OUTFD_CONV].fTorque	:=	 gDevice.stMachineDevices.aDriveInterfaces[E_DRIVE_Name.OUTFD_CONV].Q.rTorque;
gHMI.aG120StatusHMI[E_DRIVE_Name.OUTFD_CONV].bTorqueLimitReached		:=  gDevice.stMachineDevices.aDriveInterfaces[E_DRIVE_Name.OUTFD_CONV].Q.stExt.xTorqueLimitReached;
gHMI.aG120StatusHMI[E_DRIVE_Name.OUTFD_CONV].bMotorOverTemp	:=  gDevice.stMachineDevices.aDriveInterfaces[E_DRIVE_Name.OUTFD_CONV].Q.stExt.xMotorOverTemp;
gHMI.aG120StatusHMI[E_DRIVE_Name.OUTFD_CONV].bHoldingBrake	:=	gDevice.stMachineDevices.aDriveInterfaces[E_DRIVE_Name.OUTFD_CONV].Q.stExt.xHoldingBrake;

IF  gDevice.stMachineDevices.aDriveInterfaces[E_DRIVE_Name.OUTFD_CONV].Q.xFault THEN

	gHMI.aG120StatusHMI[E_DRIVE_Name.OUTFD_CONV].eDriveStatus			:= E_DRIVE_ERROR;

ELSIF gDevice.stMachineDevices.aDriveInterfaces[E_DRIVE_Name.OUTFD_CONV].Q.rActualSpeed > 0 THEN

	gHMI.aG120StatusHMI[E_DRIVE_Name.OUTFD_CONV].eDriveStatus			:= E_DRIVE_RUNING;
ELSE
	gHMI.aG120StatusHMI[E_DRIVE_Name.OUTFD_CONV].eDriveStatus			:= E_DRIVE_SPOPPED;
END_IF
END_ACTION

ACTION Init:
gDevice.stMachineDevices.aPNetMasterStatus[1].nPNetIoError := nNoCheckPNetIoError;


gDevice.stMachineDevices.aDriveInterfaces[E_DRIVE_Name.OUTER_SEPAR].I.stExt.rReferenceSpeedFrequencyP2000 := 3000;
gDevice.stMachineDevices.aDriveInterfaces[E_DRIVE_Name.OUTER_SEPAR].I.stExt.rReferenceCurrentP2002 := 5;
gDevice.stMachineDevices.aDriveInterfaces[E_DRIVE_Name.OUTER_SEPAR].I.stExt.rReferenceTorqueP2003 := 1.64;
gDevice.stMachineDevices.aDriveInterfaces[E_DRIVE_Name.OUTER_SEPAR].I.stExt.rSpeedScalefactor := 155;
gDevice.stMachineDevices.aDriveInterfaces[E_DRIVE_Name.OUTER_SEPAR].I.stExt.rTorqueScaleFactor  := 120.48;
gDevice.stMachineDevices.aDriveInterfaces[E_DRIVE_Name.OUTER_SEPAR].I.stExt.tRumpUpTime	 := T#1S;


gDevice.stMachineDevices.aDriveInterfaces[E_DRIVE_Name.INFEED_CONV].I.stExt.rReferenceSpeedFrequencyP2000 := 3000;
gDevice.stMachineDevices.aDriveInterfaces[E_DRIVE_Name.INFEED_CONV].I.stExt.rReferenceCurrentP2002 := 5;
gDevice.stMachineDevices.aDriveInterfaces[E_DRIVE_Name.INFEED_CONV].I.stExt.rReferenceTorqueP2003 := 2.46;
gDevice.stMachineDevices.aDriveInterfaces[E_DRIVE_Name.INFEED_CONV].I.stExt.rSpeedScalefactor := 155;
gDevice.stMachineDevices.aDriveInterfaces[E_DRIVE_Name.INFEED_CONV].I.stExt.rTorqueScaleFactor  := 120.48;
gDevice.stMachineDevices.aDriveInterfaces[E_DRIVE_Name.INFEED_CONV].I.stExt.tRumpUpTime	 := t#1s;


gDevice.stMachineDevices.aDriveInterfaces[E_DRIVE_Name.ROTARY_TRNSFR].I.stExt.rReferenceSpeedFrequencyP2000 := 3000;
gDevice.stMachineDevices.aDriveInterfaces[E_DRIVE_Name.ROTARY_TRNSFR].I.stExt.rReferenceCurrentP2002 := 5;
gDevice.stMachineDevices.aDriveInterfaces[E_DRIVE_Name.ROTARY_TRNSFR].I.stExt.rReferenceTorqueP2003 := 2.5;
gDevice.stMachineDevices.aDriveInterfaces[E_DRIVE_Name.ROTARY_TRNSFR].I.stExt.rSpeedScalefactor := 155;
gDevice.stMachineDevices.aDriveInterfaces[E_DRIVE_Name.ROTARY_TRNSFR].I.stExt.rTorqueScaleFactor  := 120.48;
gDevice.stMachineDevices.aDriveInterfaces[E_DRIVE_Name.ROTARY_TRNSFR].I.stExt.tRumpUpTime	 := t#1s;


gDevice.stMachineDevices.aDriveInterfaces[E_DRIVE_Name.LOWR_BELTS].I.stExt.rReferenceSpeedFrequencyP2000 := 3000;
gDevice.stMachineDevices.aDriveInterfaces[E_DRIVE_Name.LOWR_BELTS].I.stExt.rReferenceCurrentP2002 := 5;
gDevice.stMachineDevices.aDriveInterfaces[E_DRIVE_Name.LOWR_BELTS].I.stExt.rReferenceTorqueP2003 := 7.32;
gDevice.stMachineDevices.aDriveInterfaces[E_DRIVE_Name.LOWR_BELTS].I.stExt.rSpeedScalefactor := 155;
gDevice.stMachineDevices.aDriveInterfaces[E_DRIVE_Name.LOWR_BELTS].I.stExt.rTorqueScaleFactor  := 120.48;
gDevice.stMachineDevices.aDriveInterfaces[E_DRIVE_Name.LOWR_BELTS].I.stExt.tRumpUpTime	 := t#1s;


gDevice.stMachineDevices.aDriveInterfaces[E_DRIVE_Name.REJECT_CONV].I.stExt.rReferenceSpeedFrequencyP2000 := 3000;
gDevice.stMachineDevices.aDriveInterfaces[E_DRIVE_Name.REJECT_CONV].I.stExt.rReferenceCurrentP2002 := 5;
gDevice.stMachineDevices.aDriveInterfaces[E_DRIVE_Name.REJECT_CONV].I.stExt.rReferenceTorqueP2003 := 1.66;
gDevice.stMachineDevices.aDriveInterfaces[E_DRIVE_Name.REJECT_CONV].I.stExt.rSpeedScalefactor := 155;
gDevice.stMachineDevices.aDriveInterfaces[E_DRIVE_Name.REJECT_CONV].I.stExt.rTorqueScaleFactor  := 120.48;
gDevice.stMachineDevices.aDriveInterfaces[E_DRIVE_Name.REJECT_CONV].I.stExt.tRumpUpTime	 := t#1s;

(*
gDevice.stMachineDevices.aDriveInterfaces[E_DRIVE_Function.TRANSF_CONV].I.stExt.rReferenceSpeedFrequencyP2000 := 1500;
gDevice.stMachineDevices.aDriveInterfaces[E_DRIVE_Function.TRANSF_CONV].I.stExt.rReferenceCurrentP2002 := 0.5;
gDevice.stMachineDevices.aDriveInterfaces[E_DRIVE_Function.TRANSF_CONV].I.stExt.rReferenceTorqueP2003 := 1.32;
gDevice.stMachineDevices.aDriveInterfaces[E_DRIVE_Function.TRANSF_CONV].I.stExt.rSpeedScalefactor := 155;
gDevice.stMachineDevices.aDriveInterfaces[E_DRIVE_Function.TRANSF_CONV].I.stExt.rTorqueScaleFactor  := 120.48;
gDevice.stMachineDevices.aDriveInterfaces[E_DRIVE_Function.TRANSF_CONV].I.stExt.tRumpUpTime	 := t#1s;


gDevice.stMachineDevices.aDriveInterfaces[E_DRIVE_Function.ADDIT_CONV].I.stExt.rReferenceSpeedFrequencyP2000 := 3000;
gDevice.stMachineDevices.aDriveInterfaces[E_DRIVE_Function.ADDIT_CONV].I.stExt.rReferenceCurrentP2002 := 5;
gDevice.stMachineDevices.aDriveInterfaces[E_DRIVE_Function.ADDIT_CONV].I.stExt.rReferenceTorqueP2003 := 5;
gDevice.stMachineDevices.aDriveInterfaces[E_DRIVE_Function.ADDIT_CONV].I.stExt.rSpeedScalefactor := 155;
gDevice.stMachineDevices.aDriveInterfaces[E_DRIVE_Function.ADDIT_CONV].I.stExt.rTorqueScaleFactor  := 120.48;
gDevice.stMachineDevices.aDriveInterfaces[E_DRIVE_Function.ADDIT_CONV].I.stExt.tRumpUpTime	 := t#1s;


gDevice.stMachineDevices.aDriveInterfaces[E_DRIVE_Function.OUTFD_CONV].I.stExt.rReferenceSpeedFrequencyP2000 := 1500;
gDevice.stMachineDevices.aDriveInterfaces[E_DRIVE_Function.OUTFD_CONV].I.stExt.rReferenceCurrentP2002 := 0.5;
gDevice.stMachineDevices.aDriveInterfaces[E_DRIVE_Function.OUTFD_CONV].I.stExt.rReferenceTorqueP2003 := 1.32;
gDevice.stMachineDevices.aDriveInterfaces[E_DRIVE_Function.OUTFD_CONV].I.stExt.rSpeedScalefactor := 155;
gDevice.stMachineDevices.aDriveInterfaces[E_DRIVE_Function.OUTFD_CONV].I.stExt.rTorqueScaleFactor  := 120.48;
gDevice.stMachineDevices.aDriveInterfaces[E_DRIVE_Function.OUTFD_CONV].I.stExt.tRumpUpTime	 := t#1s;*)


gDevice.stMachineDevices.aDriveInterfaces[E_DRIVE_Name.TRANSF_CONV].I.stExt.rReferenceSpeedFrequencyP2000 := 3000;
gDevice.stMachineDevices.aDriveInterfaces[E_DRIVE_Name.TRANSF_CONV].I.stExt.rReferenceCurrentP2002 := 5;
gDevice.stMachineDevices.aDriveInterfaces[E_DRIVE_Name.TRANSF_CONV].I.stExt.rReferenceTorqueP2003 := 10;
gDevice.stMachineDevices.aDriveInterfaces[E_DRIVE_Name.TRANSF_CONV].I.stExt.rSpeedScalefactor := 155;
gDevice.stMachineDevices.aDriveInterfaces[E_DRIVE_Name.TRANSF_CONV].I.stExt.rTorqueScaleFactor  := 120.48;
gDevice.stMachineDevices.aDriveInterfaces[E_DRIVE_Name.TRANSF_CONV].I.stExt.tRumpUpTime	 := t#1s;


gDevice.stMachineDevices.aDriveInterfaces[E_DRIVE_Name.ADDIT_CONV].I.stExt.rReferenceSpeedFrequencyP2000 := 3000;
gDevice.stMachineDevices.aDriveInterfaces[E_DRIVE_Name.ADDIT_CONV].I.stExt.rReferenceCurrentP2002 := 5;
gDevice.stMachineDevices.aDriveInterfaces[E_DRIVE_Name.ADDIT_CONV].I.stExt.rReferenceTorqueP2003 := 10;
gDevice.stMachineDevices.aDriveInterfaces[E_DRIVE_Name.ADDIT_CONV].I.stExt.rSpeedScalefactor := 155;
gDevice.stMachineDevices.aDriveInterfaces[E_DRIVE_Name.ADDIT_CONV].I.stExt.rTorqueScaleFactor  := 120.48;
gDevice.stMachineDevices.aDriveInterfaces[E_DRIVE_Name.ADDIT_CONV].I.stExt.tRumpUpTime	 := T#1S;


gDevice.stMachineDevices.aDriveInterfaces[E_DRIVE_Name.OUTFD_CONV].I.stExt.rReferenceSpeedFrequencyP2000 := 3000;
gDevice.stMachineDevices.aDriveInterfaces[E_DRIVE_Name.OUTFD_CONV].I.stExt.rReferenceCurrentP2002 := 5;
gDevice.stMachineDevices.aDriveInterfaces[E_DRIVE_Name.OUTFD_CONV].I.stExt.rReferenceTorqueP2003 := 10;
gDevice.stMachineDevices.aDriveInterfaces[E_DRIVE_Name.OUTFD_CONV].I.stExt.rSpeedScalefactor := 155;
gDevice.stMachineDevices.aDriveInterfaces[E_DRIVE_Name.OUTFD_CONV].I.stExt.rTorqueScaleFactor  := 120.48;
gDevice.stMachineDevices.aDriveInterfaces[E_DRIVE_Name.OUTFD_CONV].I.stExt.tRumpUpTime	 := t#1s;
END_ACTION

ACTION InitConfig:
gDevice.stMachineDevices.aPNetMasterStatus[1].nPNetIoError := nNoCheckPNetIoError;


gDevice.stMachineDevices.aDriveInterfaces[E_DRIVE_Name.OUTER_SEPAR].I.stExt.rReferenceSpeedFrequencyP2000 := gDevice.stMachineConfig.aProfiNetDrive[E_DRIVE_Name.OUTER_SEPAR].fReferenceSpeedFrequencyP2000;
gDevice.stMachineDevices.aDriveInterfaces[E_DRIVE_Name.OUTER_SEPAR].I.stExt.rReferenceCurrentP2002 := gDevice.stMachineConfig.aProfiNetDrive[E_DRIVE_Name.OUTER_SEPAR].fReferenceCurrentP2002;
gDevice.stMachineDevices.aDriveInterfaces[E_DRIVE_Name.OUTER_SEPAR].I.stExt.rReferenceTorqueP2003 :=gDevice.stMachineConfig.aProfiNetDrive[E_DRIVE_Name.OUTER_SEPAR].fReferenceTorqueP2003;
gDevice.stMachineDevices.aDriveInterfaces[E_DRIVE_Name.OUTER_SEPAR].I.stExt.rSpeedScalefactor := gDevice.stMachineConfig.aProfiNetDrive[E_DRIVE_Name.OUTER_SEPAR].fSpeedScalefactor;
gDevice.stMachineDevices.aDriveInterfaces[E_DRIVE_Name.OUTER_SEPAR].I.stExt.rTorqueScaleFactor  := gDevice.stMachineConfig.aProfiNetDrive[E_DRIVE_Name.OUTER_SEPAR].fTorqueScaleFactor;
gDevice.stMachineDevices.aDriveInterfaces[E_DRIVE_Name.OUTER_SEPAR].I.stExt.tRumpUpTime	 := gDevice.stMachineConfig.aProfiNetDrive[E_DRIVE_Name.OUTER_SEPAR].tRumpUpTime;


gDevice.stMachineDevices.aDriveInterfaces[E_DRIVE_Name.INFEED_CONV].I.stExt.rReferenceSpeedFrequencyP2000 := gDevice.stMachineConfig.aProfiNetDrive[E_DRIVE_Name.INFEED_CONV].fReferenceSpeedFrequencyP2000;
gDevice.stMachineDevices.aDriveInterfaces[E_DRIVE_Name.INFEED_CONV].I.stExt.rReferenceCurrentP2002 := gDevice.stMachineConfig.aProfiNetDrive[E_DRIVE_Name.INFEED_CONV].fReferenceCurrentP2002;
gDevice.stMachineDevices.aDriveInterfaces[E_DRIVE_Name.INFEED_CONV].I.stExt.rReferenceTorqueP2003 :=gDevice.stMachineConfig.aProfiNetDrive[E_DRIVE_Name.INFEED_CONV].fReferenceTorqueP2003;
gDevice.stMachineDevices.aDriveInterfaces[E_DRIVE_Name.INFEED_CONV].I.stExt.rSpeedScalefactor := gDevice.stMachineConfig.aProfiNetDrive[E_DRIVE_Name.INFEED_CONV].fSpeedScalefactor;
gDevice.stMachineDevices.aDriveInterfaces[E_DRIVE_Name.INFEED_CONV].I.stExt.rTorqueScaleFactor  := gDevice.stMachineConfig.aProfiNetDrive[E_DRIVE_Name.INFEED_CONV].fTorqueScaleFactor;
gDevice.stMachineDevices.aDriveInterfaces[E_DRIVE_Name.INFEED_CONV].I.stExt.tRumpUpTime	 := gDevice.stMachineConfig.aProfiNetDrive[E_DRIVE_Name.INFEED_CONV].tRumpUpTime;


gDevice.stMachineDevices.aDriveInterfaces[E_DRIVE_Name.ROTARY_TRNSFR].I.stExt.rReferenceSpeedFrequencyP2000 := gDevice.stMachineConfig.aProfiNetDrive[E_DRIVE_Name.ROTARY_TRNSFR].fReferenceSpeedFrequencyP2000;
gDevice.stMachineDevices.aDriveInterfaces[E_DRIVE_Name.ROTARY_TRNSFR].I.stExt.rReferenceCurrentP2002 := gDevice.stMachineConfig.aProfiNetDrive[E_DRIVE_Name.ROTARY_TRNSFR].fReferenceCurrentP2002;
gDevice.stMachineDevices.aDriveInterfaces[E_DRIVE_Name.ROTARY_TRNSFR].I.stExt.rReferenceTorqueP2003 :=gDevice.stMachineConfig.aProfiNetDrive[E_DRIVE_Name.ROTARY_TRNSFR].fReferenceTorqueP2003;
gDevice.stMachineDevices.aDriveInterfaces[E_DRIVE_Name.ROTARY_TRNSFR].I.stExt.rSpeedScalefactor := gDevice.stMachineConfig.aProfiNetDrive[E_DRIVE_Name.ROTARY_TRNSFR].fSpeedScalefactor;
gDevice.stMachineDevices.aDriveInterfaces[E_DRIVE_Name.ROTARY_TRNSFR].I.stExt.rTorqueScaleFactor  := gDevice.stMachineConfig.aProfiNetDrive[E_DRIVE_Name.ROTARY_TRNSFR].fTorqueScaleFactor;
gDevice.stMachineDevices.aDriveInterfaces[E_DRIVE_Name.ROTARY_TRNSFR].I.stExt.tRumpUpTime	 := gDevice.stMachineConfig.aProfiNetDrive[E_DRIVE_Name.ROTARY_TRNSFR].tRumpUpTime;

gDevice.stMachineDevices.aDriveInterfaces[E_DRIVE_Name.LOWR_BELTS].I.stExt.rReferenceSpeedFrequencyP2000 := gDevice.stMachineConfig.aProfiNetDrive[E_DRIVE_Name.LOWR_BELTS].fReferenceSpeedFrequencyP2000;
gDevice.stMachineDevices.aDriveInterfaces[E_DRIVE_Name.LOWR_BELTS].I.stExt.rReferenceCurrentP2002 := gDevice.stMachineConfig.aProfiNetDrive[E_DRIVE_Name.LOWR_BELTS].fReferenceCurrentP2002;
gDevice.stMachineDevices.aDriveInterfaces[E_DRIVE_Name.LOWR_BELTS].I.stExt.rReferenceTorqueP2003 :=gDevice.stMachineConfig.aProfiNetDrive[E_DRIVE_Name.LOWR_BELTS].fReferenceTorqueP2003;
gDevice.stMachineDevices.aDriveInterfaces[E_DRIVE_Name.LOWR_BELTS].I.stExt.rSpeedScalefactor := gDevice.stMachineConfig.aProfiNetDrive[E_DRIVE_Name.LOWR_BELTS].fSpeedScalefactor;
gDevice.stMachineDevices.aDriveInterfaces[E_DRIVE_Name.LOWR_BELTS].I.stExt.rTorqueScaleFactor  := gDevice.stMachineConfig.aProfiNetDrive[E_DRIVE_Name.LOWR_BELTS].fTorqueScaleFactor;
gDevice.stMachineDevices.aDriveInterfaces[E_DRIVE_Name.LOWR_BELTS].I.stExt.tRumpUpTime	 := gDevice.stMachineConfig.aProfiNetDrive[E_DRIVE_Name.LOWR_BELTS].tRumpUpTime;


gDevice.stMachineDevices.aDriveInterfaces[E_DRIVE_Name.REJECT_CONV].I.stExt.rReferenceSpeedFrequencyP2000 := gDevice.stMachineConfig.aProfiNetDrive[E_DRIVE_Name.REJECT_CONV].fReferenceSpeedFrequencyP2000;
gDevice.stMachineDevices.aDriveInterfaces[E_DRIVE_Name.REJECT_CONV].I.stExt.rReferenceCurrentP2002 := gDevice.stMachineConfig.aProfiNetDrive[E_DRIVE_Name.REJECT_CONV].fReferenceCurrentP2002;
gDevice.stMachineDevices.aDriveInterfaces[E_DRIVE_Name.REJECT_CONV].I.stExt.rReferenceTorqueP2003 :=gDevice.stMachineConfig.aProfiNetDrive[E_DRIVE_Name.REJECT_CONV].fReferenceTorqueP2003;
gDevice.stMachineDevices.aDriveInterfaces[E_DRIVE_Name.REJECT_CONV].I.stExt.rSpeedScalefactor := gDevice.stMachineConfig.aProfiNetDrive[E_DRIVE_Name.REJECT_CONV].fSpeedScalefactor;
gDevice.stMachineDevices.aDriveInterfaces[E_DRIVE_Name.REJECT_CONV].I.stExt.rTorqueScaleFactor  := gDevice.stMachineConfig.aProfiNetDrive[E_DRIVE_Name.REJECT_CONV].fTorqueScaleFactor;
gDevice.stMachineDevices.aDriveInterfaces[E_DRIVE_Name.REJECT_CONV].I.stExt.tRumpUpTime	 := gDevice.stMachineConfig.aProfiNetDrive[E_DRIVE_Name.REJECT_CONV].tRumpUpTime;


gDevice.stMachineDevices.aDriveInterfaces[E_DRIVE_Name.TRANSF_CONV].I.stExt.rReferenceSpeedFrequencyP2000 := gDevice.stMachineConfig.aProfiNetDrive[E_DRIVE_Name.TRANSF_CONV].fReferenceSpeedFrequencyP2000;
gDevice.stMachineDevices.aDriveInterfaces[E_DRIVE_Name.TRANSF_CONV].I.stExt.rReferenceCurrentP2002 := gDevice.stMachineConfig.aProfiNetDrive[E_DRIVE_Name.TRANSF_CONV].fReferenceCurrentP2002;
gDevice.stMachineDevices.aDriveInterfaces[E_DRIVE_Name.TRANSF_CONV].I.stExt.rReferenceTorqueP2003 :=gDevice.stMachineConfig.aProfiNetDrive[E_DRIVE_Name.TRANSF_CONV].fReferenceTorqueP2003;
gDevice.stMachineDevices.aDriveInterfaces[E_DRIVE_Name.TRANSF_CONV].I.stExt.rSpeedScalefactor := gDevice.stMachineConfig.aProfiNetDrive[E_DRIVE_Name.TRANSF_CONV].fSpeedScalefactor;
gDevice.stMachineDevices.aDriveInterfaces[E_DRIVE_Name.TRANSF_CONV].I.stExt.rTorqueScaleFactor  := gDevice.stMachineConfig.aProfiNetDrive[E_DRIVE_Name.TRANSF_CONV].fTorqueScaleFactor;
gDevice.stMachineDevices.aDriveInterfaces[E_DRIVE_Name.TRANSF_CONV].I.stExt.tRumpUpTime	 := gDevice.stMachineConfig.aProfiNetDrive[E_DRIVE_Name.TRANSF_CONV].tRumpUpTime;


gDevice.stMachineDevices.aDriveInterfaces[E_DRIVE_Name.ADDIT_CONV].I.stExt.rReferenceSpeedFrequencyP2000 := gDevice.stMachineConfig.aProfiNetDrive[E_DRIVE_Name.ADDIT_CONV].fReferenceSpeedFrequencyP2000;
gDevice.stMachineDevices.aDriveInterfaces[E_DRIVE_Name.ADDIT_CONV].I.stExt.rReferenceCurrentP2002 := gDevice.stMachineConfig.aProfiNetDrive[E_DRIVE_Name.ADDIT_CONV].fReferenceCurrentP2002;
gDevice.stMachineDevices.aDriveInterfaces[E_DRIVE_Name.ADDIT_CONV].I.stExt.rReferenceTorqueP2003 :=gDevice.stMachineConfig.aProfiNetDrive[E_DRIVE_Name.ADDIT_CONV].fReferenceTorqueP2003;
gDevice.stMachineDevices.aDriveInterfaces[E_DRIVE_Name.ADDIT_CONV].I.stExt.rSpeedScalefactor := gDevice.stMachineConfig.aProfiNetDrive[E_DRIVE_Name.ADDIT_CONV].fSpeedScalefactor;
gDevice.stMachineDevices.aDriveInterfaces[E_DRIVE_Name.ADDIT_CONV].I.stExt.rTorqueScaleFactor  := gDevice.stMachineConfig.aProfiNetDrive[E_DRIVE_Name.ADDIT_CONV].fTorqueScaleFactor;
gDevice.stMachineDevices.aDriveInterfaces[E_DRIVE_Name.ADDIT_CONV].I.stExt.tRumpUpTime	 := gDevice.stMachineConfig.aProfiNetDrive[E_DRIVE_Name.ADDIT_CONV].tRumpUpTime;


gDevice.stMachineDevices.aDriveInterfaces[E_DRIVE_Name.OUTFD_CONV].I.stExt.rReferenceSpeedFrequencyP2000 := gDevice.stMachineConfig.aProfiNetDrive[E_DRIVE_Name.OUTFD_CONV].fReferenceSpeedFrequencyP2000;
gDevice.stMachineDevices.aDriveInterfaces[E_DRIVE_Name.OUTFD_CONV].I.stExt.rReferenceCurrentP2002 := gDevice.stMachineConfig.aProfiNetDrive[E_DRIVE_Name.OUTFD_CONV].fReferenceCurrentP2002;
gDevice.stMachineDevices.aDriveInterfaces[E_DRIVE_Name.OUTFD_CONV].I.stExt.rReferenceTorqueP2003 :=gDevice.stMachineConfig.aProfiNetDrive[E_DRIVE_Name.OUTFD_CONV].fReferenceTorqueP2003;
gDevice.stMachineDevices.aDriveInterfaces[E_DRIVE_Name.OUTFD_CONV].I.stExt.rSpeedScalefactor := gDevice.stMachineConfig.aProfiNetDrive[E_DRIVE_Name.OUTFD_CONV].fSpeedScalefactor;
gDevice.stMachineDevices.aDriveInterfaces[E_DRIVE_Name.OUTFD_CONV].I.stExt.rTorqueScaleFactor  := gDevice.stMachineConfig.aProfiNetDrive[E_DRIVE_Name.OUTFD_CONV].fTorqueScaleFactor;
gDevice.stMachineDevices.aDriveInterfaces[E_DRIVE_Name.OUTFD_CONV].I.stExt.tRumpUpTime	 := gDevice.stMachineConfig.aProfiNetDrive[E_DRIVE_Name.OUTFD_CONV].tRumpUpTime;
END_ACTION

END_PROGRAM

(* stored: Version 1.1.0.1
   POU C20_ProfinetDrivesCtrl: Id {05c97027-6493-4c00-b025-99caf788c068}, SpecialFunc None
   Action DrivesStatusInterface: Id {a3a54323-613b-4842-932f-6858db431e08}
   Action Init: Id {21f5bda3-cb34-4c7f-aa68-fc1080b8844d}
   Action InitConfig: Id {55a0482e-153a-40a0-b130-0b4305292275} *)
